(* Logix 5000 project; controller p65 vendor 1 type 14 code 85 rev 20.11; software revision 20.01 *)

TASK ACSTask (continuous, watchdog 500 ms) : Battery, Comm, DCMicroGrid, House01, House02, House03, House04, House05

MODULES
   Local : vendor 1 type 14 code 85 (ICP 4, rev 20.11)
      o : 1756-OB32 (ICP 3, rev 3.1, Output RPI 50 ms)
      i8 : 1756-IF8 (ICP 2, rev 1.1, Input RPI 100 ms)
      i16 : 1756-IF16 (ICP 1, rev 1.1, Input RPI 100 ms)
END_MODULES

VAR_GLOBAL   (* controller tags *)
   BatterybattCurrent : ALIAS FOR REAL00_0;
   BatterybattCurrentHILS : ALIAS FOR plc1_local_3[4];
   Batterybattcurrentoffset : REAL := 2.5261052;
   BatterybattCurrentRaw : ALIAS FOR Local:1:I.Ch4Data;
   BatterybattPower : ALIAS FOR REAL00_1;
   BatterybattVoltage : ALIAS FOR REAL00_2;
   BatterybattVoltageHILS : ALIAS FOR plc1_local_3[5];
   BatterybattVoltageRaw : ALIAS FOR Local:1:I.Ch0Data;
   BatterycanSupplyPower : ALIAS FOR DINT00_22.0;
   Batterycharge : ALIAS FOR REAL00_3;
   BatterychargeCurrent : ALIAS FOR REAL00_4;
   BatterychargeToGo : ALIAS FOR REAL00_5;
   BatterychargingTimer : ALIAS FOR CLTIMER00_0;
   BatterycomputeAddition : ALIAS FOR DINT00_22.7;
   BatterycomputeSubtraction : ALIAS FOR DINT00_22.8;
   BatterydecideToCharge : ALIAS FOR DINT00_22.15;
   BatterydecideToDisconnect : ALIAS FOR DINT00_22.16;
   BatterydeltaCharge : ALIAS FOR REAL00_6;
   BatterydischargeCurrent : ALIAS FOR REAL00_7;
   BatterydischargingTimer : ALIAS FOR CLTIMER00_1;
   BatterydisconnectedTimer : ALIAS FOR CLTIMER00_2;
   Batteryefficiency : ALIAS FOR REAL00_8;
   Batteryfraction : ALIAS FOR REAL00_9;
   BatteryfractionCharged : ALIAS FOR REAL00_10;
   BatteryfractionChargedEstimate : ALIAS FOR REAL00_11;
   BatteryfractionToGo : ALIAS FOR REAL00_12;
   BatteryfullCharge : ALIAS FOR REAL00_13;
   BatteryfullChargeCurrent : ALIAS FOR REAL00_14;
   BatterygeneralTimer : ALIAS FOR CLTIMER00_3;
   BatterygridCurrent : ALIAS FOR REAL00_15;
   BatterygridCurrentabs : REAL := 0.7502556;
   BatterygridCurrentHILS : ALIAS FOR plc1_local_3[2];
   Batterygridcurrentoffset : REAL := 2.529666;
   BatterygridCurrentRaw : ALIAS FOR Local:1:I.Ch5Data;
   BatterygridPower : ALIAS FOR REAL00_16;
   BatterygridVoltage : ALIAS FOR REAL00_17;
   BatterygridVoltageHILS : ALIAS FOR plc1_local_3[3];
   BatterygridVoltageRaw : ALIAS FOR Local:1:I.Ch9Data;
   BatteryintReqCharge : ALIAS FOR DINT00_22.17;
   BatteryintReqDischarge : ALIAS FOR DINT00_22.18;
   BatteryintReqDisconnect : ALIAS FOR DINT00_22.19;
   BatteryisCharging : ALIAS FOR DINT00_22.20;
   BatteryisDischarging : ALIAS FOR DINT00_22.21;
   BatteryisDisconnected : ALIAS FOR DINT00_22.22;
   BatteryisFullyCharged : ALIAS FOR DINT00_22.23;
   BatteryisFunctional : ALIAS FOR DINT00_22.24;
   BatterylastChargingTime : ALIAS FOR DINT00_0;
   BatterylastDischargingTime : ALIAS FOR DINT00_1;
   BatterylastDisconnectedTime : ALIAS FOR DINT00_2;
   BatterylastFractionChargedDelta : ALIAS FOR REAL00_18;
   BatterylastIntReqCharge : ALIAS FOR DINT00_22.25;
   BatterylastIntReqDischarge : ALIAS FOR DINT00_22.26;
   BatterylastIntReqDisconnect : ALIAS FOR DINT00_22.27;
   BatterylowestSOC : ALIAS FOR REAL00_19;
   Batterymultiplier : ALIAS FOR REAL00_20;
   BatterynominalDischargeCurrent : ALIAS FOR REAL00_21;
   BatteryocVoltage : ALIAS FOR REAL00_22;
   BatteryoutOfOperationalRange : ALIAS FOR DINT00_22.28;
   BatterypeukertLessOne : ALIAS FOR REAL00_23;
   Batteryproduct : ALIAS FOR REAL00_24;
   BatteryreqCharge : ALIAS FOR DINT00_22.29;
   BatteryreqDischarge : ALIAS FOR DINT00_22.30;
   BatteryreqDisconnect : ALIAS FOR DINT00_22.31;
   BatteryreqInitialize : ALIAS FOR DINT00_23.0;
   BatterysettlingTimer : ALIAS FOR CLTIMER00_4;
   Batterysoc : ALIAS FOR REAL00_25;
   BatterysocToGo : ALIAS FOR REAL00_26;
   BatterySOCTooLowEventFail : ALIAS FOR DINT00_23.1;
   BatterySOCTooLowEventSuccess : ALIAS FOR DINT00_23.2;
   BatterySOCTooLowFailTimer : ALIAS FOR CLTIMER00_5;
   BatterySOCTooLowInProcess : ALIAS FOR DINT00_23.3;
   BatterySOCTooLowMsg : ALIAS FOR MESSAGE00_0;
   BatterySOCTooLowSuccessTimer : ALIAS FOR CLTIMER00_6;
   BatterytimeSinceLastMeasurement : ALIAS FOR REAL00_27;
   BatterytimeToLowestSOC : ALIAS FOR REAL00_28;
   BatteryunambiguousCommand : ALIAS FOR DINT00_23.4;
   BG_SG_Relay : ALIAS FOR plc1_local_6[1].1;
   CB_SG1_Relay : ALIAS FOR plc1_local_6[1].5;
   CB_SG2_Relay : ALIAS FOR plc1_local_6[1].6;
   CBclose : ALIAS FOR Local:3:O.Data.15;
   CBcloseHILS : ALIAS FOR plc1_local_6[0].14;
   CBcloseProxy : ALIAS FOR DINT00_22.1;
   CBintReqClose : ALIAS FOR DINT00_22.2;
   CBisClosed : ALIAS FOR DINT00_22.3;
   CBisOpen : ALIAS FOR DINT00_22.4;
   CBreqClose : ALIAS FOR DINT00_22.5;
   CBreqOpen : ALIAS FOR DINT00_22.6;
   CF_SG_Relay : ALIAS FOR plc1_local_6[1].7;
   CL1_SG1_Relay : ALIAS FOR plc1_local_6[1].18;
   CL1_SG2_Relay : ALIAS FOR plc1_local_6[1].19;
   CL2_SG1_Relay : ALIAS FOR plc1_local_6[1].20;
   CL2_SG2_Relay : ALIAS FOR plc1_local_6[1].21;
   CL3_SG1_Relay : ALIAS FOR plc1_local_6[1].22;
   CL3_SG2_Relay : ALIAS FOR plc1_local_6[1].23;
   CL4_SG1_Relay : ALIAS FOR plc1_local_6[1].24;
   CL4_SG2_Relay : ALIAS FOR plc1_local_6[1].25;
   CL5_SG1_Relay : ALIAS FOR plc1_local_6[1].26;
   CL5_SG2_Relay : ALIAS FOR plc1_local_6[1].27;
   CLTIMER00_0 : TIMER := (PRE := 1000);
   CLTIMER00_1 : TIMER := (PRE := 1000);
   CLTIMER00_10 : TIMER := (PRE := 3600);
   CLTIMER00_100 : TIMER := (PRE := 1000);
   CLTIMER00_101 : TIMER := (PRE := 5000);
   CLTIMER00_102 : TIMER;
   CLTIMER00_103 : TIMER;
   CLTIMER00_104 : TIMER;
   CLTIMER00_105 : TIMER;
   CLTIMER00_106 : TIMER;
   CLTIMER00_107 : TIMER;
   CLTIMER00_108 : TIMER;
   CLTIMER00_109 : TIMER;
   CLTIMER00_11 : TIMER := (PRE := 3000);
   CLTIMER00_110 : TIMER;
   CLTIMER00_111 : TIMER;
   CLTIMER00_112 : TIMER;
   CLTIMER00_113 : TIMER;
   CLTIMER00_114 : TIMER;
   CLTIMER00_115 : TIMER;
   CLTIMER00_116 : TIMER;
   CLTIMER00_117 : TIMER;
   CLTIMER00_118 : TIMER;
   CLTIMER00_119 : TIMER;
   CLTIMER00_12 : TIMER := (PRE := 10000);
   CLTIMER00_120 : TIMER;
   CLTIMER00_121 : TIMER;
   CLTIMER00_13 : TIMER := (PRE := 5000);
   CLTIMER00_14 : TIMER := (PRE := 10000);
   CLTIMER00_15 : TIMER := (PRE := 500, ACC := 78, EN := 1, TT := 1);
   CLTIMER00_16 : TIMER := (PRE := 5000);
   CLTIMER00_17 : TIMER := (PRE := 3600);
   CLTIMER00_18 : TIMER := (PRE := 3000);
   CLTIMER00_19 : TIMER := (PRE := 10000);
   CLTIMER00_2 : TIMER := (PRE := 1000, ACC := 9, EN := 1, TT := 1);
   CLTIMER00_20 : TIMER := (PRE := 5000);
   CLTIMER00_21 : TIMER := (PRE := 10000);
   CLTIMER00_22 : TIMER := (PRE := 500, ACC := 120, EN := 1, TT := 1);
   CLTIMER00_23 : TIMER := (PRE := 5000);
   CLTIMER00_24 : TIMER := (PRE := 3600);
   CLTIMER00_25 : TIMER := (PRE := 3000);
   CLTIMER00_26 : TIMER := (PRE := 10000);
   CLTIMER00_27 : TIMER := (PRE := 5000);
   CLTIMER00_28 : TIMER := (PRE := 10000);
   CLTIMER00_29 : TIMER := (PRE := 500, ACC := 69, EN := 1, TT := 1);
   CLTIMER00_3 : TIMER := (PRE := 18000, ACC := 9391, EN := 1, TT := 1);
   CLTIMER00_30 : TIMER := (PRE := 5000);
   CLTIMER00_31 : TIMER := (PRE := 3600);
   CLTIMER00_32 : TIMER := (PRE := 3000);
   CLTIMER00_33 : TIMER := (PRE := 10000);
   CLTIMER00_34 : TIMER := (PRE := 5000);
   CLTIMER00_35 : TIMER := (PRE := 10000);
   CLTIMER00_36 : TIMER := (PRE := 500, ACC := 65, EN := 1, TT := 1);
   CLTIMER00_37 : TIMER := (PRE := 5000);
   CLTIMER00_38 : TIMER := (PRE := 3600);
   CLTIMER00_39 : TIMER := (PRE := 3000);
   CLTIMER00_4 : TIMER := (PRE := 300000, ACC := 17125, EN := 1, TT := 1);
   CLTIMER00_40 : TIMER := (PRE := 10000);
   CLTIMER00_41 : TIMER := (PRE := 5000);
   CLTIMER00_42 : TIMER := (PRE := 10000);
   CLTIMER00_43 : TIMER := (PRE := 500, ACC := 121, EN := 1, TT := 1);
   CLTIMER00_44 : TIMER := (PRE := 60000);
   CLTIMER00_45 : TIMER := (PRE := 1000);
   CLTIMER00_46 : TIMER := (PRE := 60000);
   CLTIMER00_47 : TIMER := (PRE := 10000, ACC := 9218, EN := 1, TT := 1);
   CLTIMER00_48 : TIMER := (PRE := 1000000);
   CLTIMER00_49 : TIMER := (PRE := 5000);
   CLTIMER00_5 : TIMER := (PRE := 5000);
   CLTIMER00_50 : TIMER := (PRE := 5000);
   CLTIMER00_51 : TIMER := (PRE := 3600);
   CLTIMER00_52 : TIMER := (PRE := 3000);
   CLTIMER00_53 : TIMER := (PRE := 10000);
   CLTIMER00_54 : TIMER := (PRE := 5000);
   CLTIMER00_55 : TIMER := (PRE := 10000);
   CLTIMER00_56 : TIMER := (PRE := 500, ACC := 26, EN := 1, TT := 1);
   CLTIMER00_57 : TIMER := (PRE := 5000);
   CLTIMER00_58 : TIMER := (PRE := 3600);
   CLTIMER00_59 : TIMER := (PRE := 3000);
   CLTIMER00_6 : TIMER := (PRE := 10000);
   CLTIMER00_60 : TIMER := (PRE := 10000);
   CLTIMER00_61 : TIMER := (PRE := 5000);
   CLTIMER00_62 : TIMER := (PRE := 10000);
   CLTIMER00_63 : TIMER := (PRE := 500, ACC := 62, EN := 1, TT := 1);
   CLTIMER00_64 : TIMER := (PRE := 5000);
   CLTIMER00_65 : TIMER := (PRE := 3600);
   CLTIMER00_66 : TIMER := (PRE := 3000);
   CLTIMER00_67 : TIMER := (PRE := 10000);
   CLTIMER00_68 : TIMER := (PRE := 5000);
   CLTIMER00_69 : TIMER := (PRE := 10000);
   CLTIMER00_7 : TIMER := (PRE := 1000000);
   CLTIMER00_70 : TIMER := (PRE := 500, ACC := 69, EN := 1, TT := 1);
   CLTIMER00_71 : TIMER := (PRE := 5000);
   CLTIMER00_72 : TIMER := (PRE := 3600);
   CLTIMER00_73 : TIMER := (PRE := 3000);
   CLTIMER00_74 : TIMER := (PRE := 10000);
   CLTIMER00_75 : TIMER := (PRE := 5000);
   CLTIMER00_76 : TIMER := (PRE := 10000);
   CLTIMER00_77 : TIMER := (PRE := 500, ACC := 90, EN := 1, TT := 1);
   CLTIMER00_78 : TIMER := (PRE := 5000);
   CLTIMER00_79 : TIMER := (PRE := 3600);
   CLTIMER00_8 : TIMER := (PRE := 5000);
   CLTIMER00_80 : TIMER := (PRE := 3000);
   CLTIMER00_81 : TIMER := (PRE := 10000);
   CLTIMER00_82 : TIMER := (PRE := 5000);
   CLTIMER00_83 : TIMER := (PRE := 10000);
   CLTIMER00_84 : TIMER := (PRE := 500, ACC := 107, EN := 1, TT := 1);
   CLTIMER00_85 : TIMER := (PRE := 60000);
   CLTIMER00_86 : TIMER := (PRE := 1000);
   CLTIMER00_87 : TIMER := (PRE := 60000);
   CLTIMER00_88 : TIMER := (PRE := 10000, ACC := 9235, EN := 1, TT := 1);
   CLTIMER00_89 : TIMER := (PRE := 10000, ACC := 9219, EN := 1, TT := 1);
   CLTIMER00_9 : TIMER := (PRE := 5000);
   CLTIMER00_90 : TIMER := (PRE := 2000);
   CLTIMER00_91 : TIMER := (PRE := 5000);
   CLTIMER00_92 : TIMER := (PRE := 3000);
   CLTIMER00_93 : TIMER := (PRE := 5000);
   CLTIMER00_94 : TIMER := (PRE := 60000);
   CLTIMER00_95 : TIMER := (PRE := 1000);
   CLTIMER00_96 : TIMER := (PRE := 5000);
   CLTIMER00_97 : TIMER := (PRE := 1000);
   CLTIMER00_98 : TIMER := (PRE := 5000);
   CLTIMER00_99 : TIMER := (PRE := 5000);
   Commaccum : ALIAS FOR REAL00_31;
   CommBattempt : ALIAS FOR DINT00_3;
   CommBclose : ALIAS FOR Local:3:O.Data.11;
   CommBcloseHILS : ALIAS FOR plc1_local_6[0].11;
   CommBcloseProxy : ALIAS FOR DINT00_23.12;
   CommBdeadBand : ALIAS FOR REAL00_32;
   CommBfailedToOpen : ALIAS FOR DINT00_23.13;
   CommBintForceOpen : ALIAS FOR DINT00_23.14;
   CommBintReqClose : ALIAS FOR DINT00_23.15;
   CommBisClosed : ALIAS FOR DINT00_23.16;
   CommBisOpen : ALIAS FOR DINT00_23.17;
   CommBmaxAttempts : ALIAS FOR DINT00_4;
   CommBmaxLoadCurrent : ALIAS FOR REAL00_33;
   CommBopenTimer : ALIAS FOR CLTIMER00_7;
   CommBreqClose : ALIAS FOR DINT00_23.18;
   CommBreqOpen : ALIAS FOR DINT00_23.19;
   CommBreqReset : ALIAS FOR DINT00_23.20;
   CommBretriesFailed : ALIAS FOR DINT00_23.21;
   CommBtooMuchCurrent : ALIAS FOR DINT00_23.22;
   CommBunexpectedLowCurrent : ALIAS FOR DINT00_23.23;
   CommcanNotifyUser : ALIAS FOR DINT00_23.24;
   CommcommandChanged : ALIAS FOR DINT00_23.25;
   CommcommandChangedTimer : ALIAS FOR CLTIMER00_8;
   Commcurrent : ALIAS FOR REAL00_34;
   CommcurrentHILS : ALIAS FOR plc1_local_3[8];
   CommcurrentRaw : ALIAS FOR Local:1:I.Ch10Data;
   Commdeadband : ALIAS FOR REAL00_35;
   Commdifference : ALIAS FOR REAL00_36;
   CommfailedToConnect : ALIAS FOR DINT00_23.26;
   CommfailedToDisconnect : ALIAS FOR DINT00_23.27;
   CommintReqConnect : ALIAS FOR DINT00_23.28;
   CommisConnected : ALIAS FOR DINT00_23.29;
   CommisDisconnected : ALIAS FOR DINT00_23.30;
   CommnotificationTimer : ALIAS FOR CLTIMER00_44;
   CommOverCurrentConditionEventFail : ALIAS FOR DINT00_27.13;
   CommOverCurrentConditionEventSuccess : ALIAS FOR DINT00_27.14;
   CommOverCurrentConditionFailTimer : ALIAS FOR CLTIMER00_45;
   CommOverCurrentConditionInProcess : ALIAS FOR DINT00_27.15;
   CommOverCurrentConditionMsg : ALIAS FOR MESSAGE00_11;
   CommOverCurrentConditionSuccessTimer : ALIAS FOR CLTIMER00_46;
   Commpower : ALIAS FOR REAL00_102;
   CommreqConnect : ALIAS FOR DINT00_27.16;
   CommreqDisconnect : ALIAS FOR DINT00_27.17;
   CommsampleNow : ALIAS FOR DINT00_27.18;
   CommsampleTimer : ALIAS FOR CLTIMER00_47;
   Commsuperuser : ALIAS FOR STRING00_5;
   Commtotal : ALIAS FOR REAL00_103;
   CommtotalTooLarge : ALIAS FOR DINT00_27.19;
   CommtotalTooSmall : ALIAS FOR DINT00_27.20;
   CommuserNotified : ALIAS FOR DINT00_27.21;
   Commvoltage : ALIAS FOR REAL00_104;
   CommvoltageHILS : ALIAS FOR plc1_local_3[9];
   CommvoltageRaw : ALIAS FOR Local:2:I.Ch7Data;
   DBclose : ALIAS FOR Local:3:O.Data.14;
   DBcloseHILS : ALIAS FOR plc1_local_6[0].13;
   DBcloseProxy : ALIAS FOR DINT00_22.9;
   DBintReqClose : ALIAS FOR DINT00_22.10;
   DBisClosed : ALIAS FOR DINT00_22.11;
   DBisOpen : ALIAS FOR DINT00_22.12;
   DBreqClose : ALIAS FOR DINT00_22.13;
   DBreqOpen : ALIAS FOR DINT00_22.14;
   DCMicroGridcanNotifyUser : ALIAS FOR DINT00_23.5;
   DCMicroGridfailedToShutdown : ALIAS FOR DINT00_23.6;
   DCMicroGridfailedToStartup : ALIAS FOR DINT00_23.7;
   DCMicroGridinitialPowerRate : ALIAS FOR REAL00_29;
   DCMicroGridisInOperation : ALIAS FOR DINT00_23.8;
   DCMicroGridisShutdown : ALIAS FOR DINT00_23.9;
   DCMicroGridisSimulating : ALIAS FOR DINT00_23.10;
   DCMicroGridisStarted : ALIAS FOR DINT00_23.11;
   DCMicroGridlowestSupportedPriority : ALIAS FOR DINT00_17;
   DCMicroGridmaxPowerRate : ALIAS FOR REAL00_185;
   DCMicroGridmorePowerAvailable : ALIAS FOR DINT00_32.12;
   DCMicroGridnotificationTimer : ALIAS FOR CLTIMER00_94;
   DCMicroGridpowerRate : ALIAS FOR REAL00_186;
   DCMicroGridpowerRateIncrement : REAL := 10.0;
   DCMicroGridrecruitingPhase : ALIAS FOR DINT00_18;
   DCMicroGridreqReset : ALIAS FOR DINT00_32.13;
   DCMicroGridreqShutdown : ALIAS FOR DINT00_32.14;
   DCMicroGridreqStartup : ALIAS FOR DINT00_32.15;
   DCMicroGridResetEventFail : ALIAS FOR DINT00_32.16;
   DCMicroGridResetEventSuccess : ALIAS FOR DINT00_32.17;
   DCMicroGridResetFailTimer : ALIAS FOR CLTIMER00_95;
   DCMicroGridResetInProcess : ALIAS FOR DINT00_32.18;
   DCMicroGridResetMsg : ALIAS FOR MESSAGE00_25;
   DCMicroGridResetSuccessTimer : ALIAS FOR CLTIMER00_96;
   DCMicroGridShutdownEventFail : ALIAS FOR DINT00_32.19;
   DCMicroGridShutdownEventSuccess : ALIAS FOR DINT00_32.20;
   DCMicroGridShutdownFailTimer : ALIAS FOR CLTIMER00_97;
   DCMicroGridShutdownInProcess : ALIAS FOR DINT00_32.21;
   DCMicroGridShutdownMsg : ALIAS FOR MESSAGE00_26;
   DCMicroGridShutdownSuccessTimer : ALIAS FOR CLTIMER00_98;
   DCMicroGridsourcesProvidingExcessPower : ALIAS FOR DINT00_33.7;
   DCMicroGridStartupEventFail : ALIAS FOR DINT00_33.8;
   DCMicroGridStartupEventSuccess : ALIAS FOR DINT00_33.9;
   DCMicroGridStartupFailTimer : ALIAS FOR CLTIMER00_100;
   DCMicroGridStartupInProcess : ALIAS FOR DINT00_33.10;
   DCMicroGridStartupMsg : ALIAS FOR MESSAGE00_27;
   DCMicroGridStartupSuccessTimer : ALIAS FOR CLTIMER00_101;
   DCMicroGridsuperuser : ALIAS FOR STRING00_12;
   DCMicroGridtest : ALIAS FOR REAL00_192;
   DCMicroGridtestout : ALIAS FOR REAL00_193;
   DCMicroGriduserNotified : ALIAS FOR DINT00_33.11;
   DINT00_0 : DINT;
   DINT00_1 : DINT;
   DINT00_10 : DINT;
   DINT00_11 : DINT := 3;
   DINT00_12 : DINT := 10;
   DINT00_13 : DINT := 9;
   DINT00_14 : DINT := 8;
   DINT00_15 : DINT := 7;
   DINT00_16 : DINT := 6;
   DINT00_17 : DINT := 10;
   DINT00_18 : DINT;
   DINT00_19 : DINT;
   DINT00_2 : DINT := 17;
   DINT00_20 : DINT;
   DINT00_21 : DINT;
   DINT00_22 : DINT := -842239919;
   DINT00_23 : DINT := 1225400868;
   DINT00_24 : DINT := 621626516;
   DINT00_25 : DINT := -733396144;
   DINT00_26 : DINT := -1808465328;
   DINT00_27 : DINT := 1086524740;
   DINT00_28 : DINT := 621957153;
   DINT00_29 : DINT := 621363348;
   DINT00_3 : DINT;
   DINT00_30 : DINT := -1811332527;
   DINT00_31 : DINT := 1646596688;
   DINT00_32 : DINT := -1978526464;
   DINT00_33 : DINT := 580;
   DINT00_34 : DINT;
   DINT00_35 : DINT;
   DINT00_4 : DINT := 3;
   DINT00_5 : DINT := 5;
   DINT00_6 : DINT := 4;
   DINT00_7 : DINT := 3;
   DINT00_8 : DINT := 2;
   DINT00_9 : DINT := 1;
   House01accountBalance : ALIAS FOR REAL00_115;
   House01accountDepositRate : ALIAS FOR REAL00_116;
   House01actualGridProvider : ALIAS FOR STRING00_6;
   House01Bclose : ALIAS FOR Local:3:O.Data.0;
   House01BcloseHILS : ALIAS FOR plc1_local_6[0].0;
   House01BcloseProxy : ALIAS FOR DINT00_28.9;
   House01BintReqClose : ALIAS FOR DINT00_28.10;
   House01BisClosed : ALIAS FOR DINT00_28.11;
   House01BisOpen : ALIAS FOR DINT00_28.12;
   House01BreqClose : ALIAS FOR DINT00_28.13;
   House01BreqOpen : ALIAS FOR DINT00_28.14;
   House01commandChanged : ALIAS FOR DINT00_28.15;
   House01commandChangedTimer : ALIAS FOR CLTIMER00_50;
   House01current : ALIAS FOR REAL00_117;
   House01currentHILS : ALIAS FOR plc1_local_2[0];
   House01currentRaw : ALIAS FOR Local:1:I.Ch12Data;
   House01deadband : ALIAS FOR REAL00_118;
   House01depositTimer : ALIAS FOR CLTIMER00_51;
   House01DisconnectPowerEventFail : ALIAS FOR DINT00_28.16;
   House01DisconnectPowerEventSuccess : ALIAS FOR DINT00_28.17;
   House01DisconnectPowerFailTimer : ALIAS FOR CLTIMER00_52;
   House01DisconnectPowerInProcess : ALIAS FOR DINT00_28.18;
   House01DisconnectPowerMsg : ALIAS FOR MESSAGE00_12;
   House01DisconnectPowerSuccessTimer : ALIAS FOR CLTIMER00_53;
   House01failedToConnect : ALIAS FOR DINT00_28.19;
   House01failedToDisconnect : ALIAS FOR DINT00_28.20;
   House01fundsAvailable : ALIAS FOR DINT00_28.21;
   House01incrementToAdd : ALIAS FOR REAL00_119;
   House01incrementToSubtract : ALIAS FOR REAL00_120;
   House01initialAccountBalance : ALIAS FOR REAL00_121;
   House01intReqConnect : ALIAS FOR DINT00_28.22;
   House01isConnected : ALIAS FOR DINT00_28.23;
   House01isDisconnected : ALIAS FOR DINT00_28.24;
   House01minBalance : ALIAS FOR REAL00_122;
   House01minBalanceToReconnect : ALIAS FOR REAL00_123;
   House01minTime : ALIAS FOR REAL00_124;
   House01powerRate : ALIAS FOR REAL00_125;
   House01powerRateMax : REAL := 40.0;
   House01priority : ALIAS FOR DINT00_12;
   House01PurchasePowerEventFail : ALIAS FOR DINT00_28.25;
   House01PurchasePowerEventSuccess : ALIAS FOR DINT00_28.26;
   House01PurchasePowerFailTimer : ALIAS FOR CLTIMER00_54;
   House01PurchasePowerInProcess : ALIAS FOR DINT00_28.27;
   House01PurchasePowerMsg : ALIAS FOR MESSAGE00_13;
   House01PurchasePowerSuccessTimer : ALIAS FOR CLTIMER00_55;
   House01reqConnect : ALIAS FOR DINT00_28.28;
   House01reqDisconnect : ALIAS FOR DINT00_28.29;
   House01runningOut : ALIAS FOR DINT00_28.30;
   House01spendingRate : ALIAS FOR REAL00_126;
   House01timeRemaining : ALIAS FOR REAL00_127;
   House01usageTimer : ALIAS FOR CLTIMER00_56;
   House02accountBalance : ALIAS FOR REAL00_128;
   House02accountDepositRate : ALIAS FOR REAL00_129;
   House02actualGridProvider : ALIAS FOR STRING00_7;
   House02Bclose : ALIAS FOR Local:3:O.Data.1;
   House02BcloseHILS : ALIAS FOR plc1_local_6[0].1;
   House02BcloseProxy : ALIAS FOR DINT00_28.31;
   House02BintReqClose : ALIAS FOR DINT00_29.0;
   House02BisClosed : ALIAS FOR DINT00_29.1;
   House02BisOpen : ALIAS FOR DINT00_29.2;
   House02BreqClose : ALIAS FOR DINT00_29.3;
   House02BreqOpen : ALIAS FOR DINT00_29.4;
   House02commandChanged : ALIAS FOR DINT00_29.5;
   House02commandChangedTimer : ALIAS FOR CLTIMER00_57;
   House02current : ALIAS FOR REAL00_130;
   House02currentHILS : ALIAS FOR plc1_local_2[1];
   House02currentRaw : ALIAS FOR Local:1:I.Ch13Data;
   House02deadband : ALIAS FOR REAL00_131;
   House02depositTimer : ALIAS FOR CLTIMER00_58;
   House02DisconnectPowerEventFail : ALIAS FOR DINT00_29.6;
   House02DisconnectPowerEventSuccess : ALIAS FOR DINT00_29.7;
   House02DisconnectPowerFailTimer : ALIAS FOR CLTIMER00_59;
   House02DisconnectPowerInProcess : ALIAS FOR DINT00_29.8;
   House02DisconnectPowerMsg : ALIAS FOR MESSAGE00_14;
   House02DisconnectPowerSuccessTimer : ALIAS FOR CLTIMER00_60;
   House02failedToConnect : ALIAS FOR DINT00_29.9;
   House02failedToDisconnect : ALIAS FOR DINT00_29.10;
   House02fundsAvailable : ALIAS FOR DINT00_29.11;
   House02incrementToAdd : ALIAS FOR REAL00_132;
   House02incrementToSubtract : ALIAS FOR REAL00_133;
   House02initialAccountBalance : ALIAS FOR REAL00_134;
   House02intReqConnect : ALIAS FOR DINT00_29.12;
   House02isConnected : ALIAS FOR DINT00_29.13;
   House02isDisconnected : ALIAS FOR DINT00_29.14;
   House02minBalance : ALIAS FOR REAL00_135;
   House02minBalanceToReconnect : ALIAS FOR REAL00_136;
   House02minTime : ALIAS FOR REAL00_137;
   House02powerRate : ALIAS FOR REAL00_138;
   House02powerRateMax : REAL := 40.0;
   House02priority : ALIAS FOR DINT00_13;
   House02PurchasePowerEventFail : ALIAS FOR DINT00_29.15;
   House02PurchasePowerEventSuccess : ALIAS FOR DINT00_29.16;
   House02PurchasePowerFailTimer : ALIAS FOR CLTIMER00_61;
   House02PurchasePowerInProcess : ALIAS FOR DINT00_29.17;
   House02PurchasePowerMsg : ALIAS FOR MESSAGE00_15;
   House02PurchasePowerSuccessTimer : ALIAS FOR CLTIMER00_62;
   House02reqConnect : ALIAS FOR DINT00_29.18;
   House02reqDisconnect : ALIAS FOR DINT00_29.19;
   House02runningOut : ALIAS FOR DINT00_29.20;
   House02spendingRate : ALIAS FOR REAL00_139;
   House02timeRemaining : ALIAS FOR REAL00_140;
   House02usageTimer : ALIAS FOR CLTIMER00_63;
   House03accountBalance : ALIAS FOR REAL00_141;
   House03accountDepositRate : ALIAS FOR REAL00_142;
   House03actualGridProvider : ALIAS FOR STRING00_8;
   House03Bclose : ALIAS FOR Local:3:O.Data.2;
   House03BcloseHILS : ALIAS FOR plc1_local_6[0].2;
   House03BcloseProxy : ALIAS FOR DINT00_29.21;
   House03BintReqClose : ALIAS FOR DINT00_29.22;
   House03BisClosed : ALIAS FOR DINT00_29.23;
   House03BisOpen : ALIAS FOR DINT00_29.24;
   House03BreqClose : ALIAS FOR DINT00_29.25;
   House03BreqOpen : ALIAS FOR DINT00_29.26;
   House03commandChanged : ALIAS FOR DINT00_29.27;
   House03commandChangedTimer : ALIAS FOR CLTIMER00_64;
   House03current : ALIAS FOR REAL00_143;
   House03currentHILS : ALIAS FOR plc1_local_2[2];
   House03currentRaw : ALIAS FOR Local:1:I.Ch14Data;
   House03deadband : ALIAS FOR REAL00_144;
   House03depositTimer : ALIAS FOR CLTIMER00_65;
   House03DisconnectPowerEventFail : ALIAS FOR DINT00_29.28;
   House03DisconnectPowerEventSuccess : ALIAS FOR DINT00_29.29;
   House03DisconnectPowerFailTimer : ALIAS FOR CLTIMER00_66;
   House03DisconnectPowerInProcess : ALIAS FOR DINT00_29.30;
   House03DisconnectPowerMsg : ALIAS FOR MESSAGE00_16;
   House03DisconnectPowerSuccessTimer : ALIAS FOR CLTIMER00_67;
   House03failedToConnect : ALIAS FOR DINT00_29.31;
   House03failedToDisconnect : ALIAS FOR DINT00_30.0;
   House03fundsAvailable : ALIAS FOR DINT00_30.1;
   House03incrementToAdd : ALIAS FOR REAL00_145;
   House03incrementToSubtract : ALIAS FOR REAL00_146;
   House03initialAccountBalance : ALIAS FOR REAL00_147;
   House03intReqConnect : ALIAS FOR DINT00_30.2;
   House03isConnected : ALIAS FOR DINT00_30.3;
   House03isDisconnected : ALIAS FOR DINT00_30.4;
   House03minBalance : ALIAS FOR REAL00_148;
   House03minBalanceToReconnect : ALIAS FOR REAL00_149;
   House03minTime : ALIAS FOR REAL00_150;
   House03powerRate : ALIAS FOR REAL00_151;
   House03powerRateMax : REAL := 30.0;
   House03priority : ALIAS FOR DINT00_14;
   House03PurchasePowerEventFail : ALIAS FOR DINT00_30.5;
   House03PurchasePowerEventSuccess : ALIAS FOR DINT00_30.6;
   House03PurchasePowerFailTimer : ALIAS FOR CLTIMER00_68;
   House03PurchasePowerInProcess : ALIAS FOR DINT00_30.7;
   House03PurchasePowerMsg : ALIAS FOR MESSAGE00_17;
   House03PurchasePowerSuccessTimer : ALIAS FOR CLTIMER00_69;
   House03reqConnect : ALIAS FOR DINT00_30.8;
   House03reqDisconnect : ALIAS FOR DINT00_30.9;
   House03runningOut : ALIAS FOR DINT00_30.10;
   House03spendingRate : ALIAS FOR REAL00_152;
   House03timeRemaining : ALIAS FOR REAL00_153;
   House03usageTimer : ALIAS FOR CLTIMER00_70;
   House04accountBalance : ALIAS FOR REAL00_154;
   House04accountDepositRate : ALIAS FOR REAL00_155;
   House04actualGridProvider : ALIAS FOR STRING00_9;
   House04Bclose : ALIAS FOR Local:3:O.Data.3;
   House04BcloseHILS : ALIAS FOR plc1_local_6[0].3;
   House04BcloseProxy : ALIAS FOR DINT00_30.11;
   House04BintReqClose : ALIAS FOR DINT00_30.12;
   House04BisClosed : ALIAS FOR DINT00_30.13;
   House04BisOpen : ALIAS FOR DINT00_30.14;
   House04BreqClose : ALIAS FOR DINT00_30.15;
   House04BreqOpen : ALIAS FOR DINT00_30.16;
   House04commandChanged : ALIAS FOR DINT00_30.17;
   House04commandChangedTimer : ALIAS FOR CLTIMER00_71;
   House04current : ALIAS FOR REAL00_156;
   House04currentHILS : ALIAS FOR plc1_local_2[3];
   House04currentRaw : ALIAS FOR Local:1:I.Ch15Data;
   House04deadband : ALIAS FOR REAL00_157;
   House04depositTimer : ALIAS FOR CLTIMER00_72;
   House04DisconnectPowerEventFail : ALIAS FOR DINT00_30.18;
   House04DisconnectPowerEventSuccess : ALIAS FOR DINT00_30.19;
   House04DisconnectPowerFailTimer : ALIAS FOR CLTIMER00_73;
   House04DisconnectPowerInProcess : ALIAS FOR DINT00_30.20;
   House04DisconnectPowerMsg : ALIAS FOR MESSAGE00_18;
   House04DisconnectPowerSuccessTimer : ALIAS FOR CLTIMER00_74;
   House04failedToConnect : ALIAS FOR DINT00_30.21;
   House04failedToDisconnect : ALIAS FOR DINT00_30.22;
   House04fundsAvailable : ALIAS FOR DINT00_30.23;
   House04incrementToAdd : ALIAS FOR REAL00_158;
   House04incrementToSubtract : ALIAS FOR REAL00_159;
   House04initialAccountBalance : ALIAS FOR REAL00_160;
   House04intReqConnect : ALIAS FOR DINT00_30.24;
   House04isConnected : ALIAS FOR DINT00_30.25;
   House04isDisconnected : ALIAS FOR DINT00_30.26;
   House04minBalance : ALIAS FOR REAL00_161;
   House04minBalanceToReconnect : ALIAS FOR REAL00_162;
   House04minTime : ALIAS FOR REAL00_163;
   House04poweRateMax : REAL;
   House04powerRate : ALIAS FOR REAL00_164;
   House04powerRateMax : REAL := 30.0;
   House04priority : ALIAS FOR DINT00_15;
   House04PurchasePowerEventFail : ALIAS FOR DINT00_30.27;
   House04PurchasePowerEventSuccess : ALIAS FOR DINT00_30.28;
   House04PurchasePowerFailTimer : ALIAS FOR CLTIMER00_75;
   House04PurchasePowerInProcess : ALIAS FOR DINT00_30.29;
   House04PurchasePowerMsg : ALIAS FOR MESSAGE00_19;
   House04PurchasePowerSuccessTimer : ALIAS FOR CLTIMER00_76;
   House04reqConnect : ALIAS FOR DINT00_30.30;
   House04reqDisconnect : ALIAS FOR DINT00_30.31;
   House04runningOut : ALIAS FOR DINT00_31.0;
   House04spendingRate : ALIAS FOR REAL00_165;
   House04timeRemaining : ALIAS FOR REAL00_166;
   House04usageTimer : ALIAS FOR CLTIMER00_77;
   House05accountBalance : ALIAS FOR REAL00_167;
   House05accountDepositRate : ALIAS FOR REAL00_168;
   House05actualGridProvider : ALIAS FOR STRING00_10;
   House05Bclose : ALIAS FOR Local:3:O.Data.4;
   House05BcloseHILS : ALIAS FOR plc1_local_6[0].4;
   House05BcloseProxy : ALIAS FOR DINT00_31.1;
   House05BintReqClose : ALIAS FOR DINT00_31.2;
   House05BisClosed : ALIAS FOR DINT00_31.3;
   House05BisOpen : ALIAS FOR DINT00_31.4;
   House05BreqClose : ALIAS FOR DINT00_31.5;
   House05BreqOpen : ALIAS FOR DINT00_31.6;
   House05commandChanged : ALIAS FOR DINT00_31.7;
   House05commandChangedTimer : ALIAS FOR CLTIMER00_78;
   House05current : ALIAS FOR REAL00_169;
   House05currentHILS : ALIAS FOR plc1_local_2[4];
   House05currentRaw : ALIAS FOR Local:2:I.Ch0Data;
   House05deadband : ALIAS FOR REAL00_170;
   House05depositTimer : ALIAS FOR CLTIMER00_79;
   House05DisconnectPowerEventFail : ALIAS FOR DINT00_31.8;
   House05DisconnectPowerEventSuccess : ALIAS FOR DINT00_31.9;
   House05DisconnectPowerFailTimer : ALIAS FOR CLTIMER00_80;
   House05DisconnectPowerInProcess : ALIAS FOR DINT00_31.10;
   House05DisconnectPowerMsg : ALIAS FOR MESSAGE00_20;
   House05DisconnectPowerSuccessTimer : ALIAS FOR CLTIMER00_81;
   House05failedToConnect : ALIAS FOR DINT00_31.11;
   House05failedToDisconnect : ALIAS FOR DINT00_31.12;
   House05fundsAvailable : ALIAS FOR DINT00_31.13;
   House05incrementToAdd : ALIAS FOR REAL00_171;
   House05incrementToSubtract : ALIAS FOR REAL00_172;
   House05initialAccountBalance : ALIAS FOR REAL00_173;
   House05intReqConnect : ALIAS FOR DINT00_31.14;
   House05isConnected : ALIAS FOR DINT00_31.15;
   House05isDisconnected : ALIAS FOR DINT00_31.16;
   House05minBalance : ALIAS FOR REAL00_174;
   House05minBalanceToReconnect : ALIAS FOR REAL00_175;
   House05minTime : ALIAS FOR REAL00_176;
   House05powerRate : ALIAS FOR REAL00_177;
   House05powerRateMax : REAL := 60.0;
   House05priority : ALIAS FOR DINT00_16;
   House05PurchasePowerEventFail : ALIAS FOR DINT00_31.17;
   House05PurchasePowerEventSuccess : ALIAS FOR DINT00_31.18;
   House05PurchasePowerFailTimer : ALIAS FOR CLTIMER00_82;
   House05PurchasePowerInProcess : ALIAS FOR DINT00_31.19;
   House05PurchasePowerMsg : ALIAS FOR MESSAGE00_21;
   House05PurchasePowerSuccessTimer : ALIAS FOR CLTIMER00_83;
   House05reqConnect : ALIAS FOR DINT00_31.20;
   House05reqDisconnect : ALIAS FOR DINT00_31.21;
   House05runningOut : ALIAS FOR DINT00_31.22;
   House05spendingRate : ALIAS FOR REAL00_178;
   House05timeRemaining : ALIAS FOR REAL00_179;
   House05usageTimer : ALIAS FOR CLTIMER00_84;
   LastSolar_Power : REAL;
   Load01accountBalance : ALIAS FOR REAL00_37;
   Load01accountDepositRate : ALIAS FOR REAL00_38;
   Load01actualGridProvider : ALIAS FOR STRING00_0;
   Load01Bclose : ALIAS FOR Local:3:O.Data.5;
   Load01BcloseHILS : ALIAS FOR plc1_local_6[0].5;
   Load01BcloseProxy : ALIAS FOR DINT00_23.31;
   Load01BintReqClose : ALIAS FOR DINT00_24.0;
   Load01BisClosed : ALIAS FOR DINT00_24.1;
   Load01BisOpen : ALIAS FOR DINT00_24.2;
   Load01BreqClose : ALIAS FOR DINT00_24.3;
   Load01BreqOpen : ALIAS FOR DINT00_24.4;
   Load01commandChanged : ALIAS FOR DINT00_24.5;
   Load01commandChangedTimer : ALIAS FOR CLTIMER00_9;
   Load01current : ALIAS FOR REAL00_39;
   Load01currentHILS : ALIAS FOR plc1_local_2[5];
   Load01currentRaw : ALIAS FOR Local:2:I.Ch2Data;
   Load01deadband : ALIAS FOR REAL00_40;
   Load01depositTimer : ALIAS FOR CLTIMER00_10;
   Load01DisconnectPowerEventFail : ALIAS FOR DINT00_24.6;
   Load01DisconnectPowerEventSuccess : ALIAS FOR DINT00_24.7;
   Load01DisconnectPowerFailTimer : ALIAS FOR CLTIMER00_11;
   Load01DisconnectPowerInProcess : ALIAS FOR DINT00_24.8;
   Load01DisconnectPowerMsg : ALIAS FOR MESSAGE00_1;
   Load01DisconnectPowerSuccessTimer : ALIAS FOR CLTIMER00_12;
   Load01failedToConnect : ALIAS FOR DINT00_24.9;
   Load01failedToDisconnect : ALIAS FOR DINT00_24.10;
   Load01fundsAvailable : ALIAS FOR DINT00_24.11;
   Load01incrementToAdd : ALIAS FOR REAL00_41;
   Load01incrementToSubtract : ALIAS FOR REAL00_42;
   Load01initialAccountBalance : ALIAS FOR REAL00_43;
   Load01intReqConnect : ALIAS FOR DINT00_24.12;
   Load01isConnected : ALIAS FOR DINT00_24.13;
   Load01isDisconnected : ALIAS FOR DINT00_24.14;
   Load01minBalance : ALIAS FOR REAL00_44;
   Load01minBalanceToReconnect : ALIAS FOR REAL00_45;
   Load01minTime : ALIAS FOR REAL00_46;
   Load01powerRate : ALIAS FOR REAL00_47;
   Load01powerRateMax : REAL := 80.0;
   Load01priority : ALIAS FOR DINT00_5;
   Load01PurchasePowerEventFail : ALIAS FOR DINT00_24.15;
   Load01PurchasePowerEventSuccess : ALIAS FOR DINT00_24.16;
   Load01PurchasePowerFailTimer : ALIAS FOR CLTIMER00_13;
   Load01PurchasePowerInProcess : ALIAS FOR DINT00_24.17;
   Load01PurchasePowerMsg : ALIAS FOR MESSAGE00_2;
   Load01PurchasePowerSuccessTimer : ALIAS FOR CLTIMER00_14;
   Load01reqConnect : ALIAS FOR DINT00_24.18;
   Load01reqDisconnect : ALIAS FOR DINT00_24.19;
   Load01runningOut : ALIAS FOR DINT00_24.20;
   Load01spendingRate : ALIAS FOR REAL00_48;
   Load01timeRemaining : ALIAS FOR REAL00_49;
   Load01usageTimer : ALIAS FOR CLTIMER00_15;
   Load02accountBalance : ALIAS FOR REAL00_50;
   Load02accountDepositRate : ALIAS FOR REAL00_51;
   Load02actualGridProvider : ALIAS FOR STRING00_1;
   Load02Bclose : ALIAS FOR Local:3:O.Data.6;
   Load02BcloseHILS : ALIAS FOR plc1_local_6[0].6;
   Load02BcloseProxy : ALIAS FOR DINT00_24.21;
   Load02BintReqClose : ALIAS FOR DINT00_24.22;
   Load02BisClosed : ALIAS FOR DINT00_24.23;
   Load02BisOpen : ALIAS FOR DINT00_24.24;
   Load02BreqClose : ALIAS FOR DINT00_24.25;
   Load02BreqOpen : ALIAS FOR DINT00_24.26;
   Load02commandChanged : ALIAS FOR DINT00_24.27;
   Load02commandChangedTimer : ALIAS FOR CLTIMER00_16;
   Load02current : ALIAS FOR REAL00_52;
   Load02currentHILS : ALIAS FOR plc1_local_2[6];
   Load02currentRaw : ALIAS FOR Local:2:I.Ch3Data;
   Load02deadband : ALIAS FOR REAL00_53;
   Load02depositTimer : ALIAS FOR CLTIMER00_17;
   Load02DisconnectPowerEventFail : ALIAS FOR DINT00_24.28;
   Load02DisconnectPowerEventSuccess : ALIAS FOR DINT00_24.29;
   Load02DisconnectPowerFailTimer : ALIAS FOR CLTIMER00_18;
   Load02DisconnectPowerInProcess : ALIAS FOR DINT00_24.30;
   Load02DisconnectPowerMsg : ALIAS FOR MESSAGE00_3;
   Load02DisconnectPowerSuccessTimer : ALIAS FOR CLTIMER00_19;
   Load02failedToConnect : ALIAS FOR DINT00_24.31;
   Load02failedToDisconnect : ALIAS FOR DINT00_25.0;
   Load02fundsAvailable : ALIAS FOR DINT00_25.1;
   Load02incrementToAdd : ALIAS FOR REAL00_54;
   Load02incrementToSubtract : ALIAS FOR REAL00_55;
   Load02initialAccountBalance : ALIAS FOR REAL00_56;
   Load02intReqConnect : ALIAS FOR DINT00_25.2;
   Load02isConnected : ALIAS FOR DINT00_25.3;
   Load02isDisconnected : ALIAS FOR DINT00_25.4;
   Load02minBalance : ALIAS FOR REAL00_57;
   Load02minBalanceToReconnect : ALIAS FOR REAL00_58;
   Load02minTime : ALIAS FOR REAL00_59;
   Load02powerRate : ALIAS FOR REAL00_60;
   Load02powerRateMax : REAL := 110.0;
   Load02priority : ALIAS FOR DINT00_6;
   Load02PurchasePowerEventFail : ALIAS FOR DINT00_25.5;
   Load02PurchasePowerEventSuccess : ALIAS FOR DINT00_25.6;
   Load02PurchasePowerFailTimer : ALIAS FOR CLTIMER00_20;
   Load02PurchasePowerInProcess : ALIAS FOR DINT00_25.7;
   Load02PurchasePowerMsg : ALIAS FOR MESSAGE00_4;
   Load02PurchasePowerSuccessTimer : ALIAS FOR CLTIMER00_21;
   Load02reqConnect : ALIAS FOR DINT00_25.8;
   Load02reqDisconnect : ALIAS FOR DINT00_25.9;
   Load02runningOut : ALIAS FOR DINT00_25.10;
   Load02spendingRate : ALIAS FOR REAL00_61;
   Load02timeRemaining : ALIAS FOR REAL00_62;
   Load02usageTimer : ALIAS FOR CLTIMER00_22;
   Load03accountBalance : ALIAS FOR REAL00_63;
   Load03accountDepositRate : ALIAS FOR REAL00_64;
   Load03actualGridProvider : ALIAS FOR STRING00_2;
   Load03Bclose : ALIAS FOR Local:3:O.Data.7;
   Load03BcloseHILS : ALIAS FOR plc1_local_6[0].7;
   Load03BcloseProxy : ALIAS FOR DINT00_25.11;
   Load03BintReqClose : ALIAS FOR DINT00_25.12;
   Load03BisClosed : ALIAS FOR DINT00_25.13;
   Load03BisOpen : ALIAS FOR DINT00_25.14;
   Load03BreqClose : ALIAS FOR DINT00_25.15;
   Load03BreqOpen : ALIAS FOR DINT00_25.16;
   Load03commandChanged : ALIAS FOR DINT00_25.17;
   Load03commandChangedTimer : ALIAS FOR CLTIMER00_23;
   Load03current : ALIAS FOR REAL00_65;
   Load03currentHILS : ALIAS FOR plc1_local_2[7];
   Load03currentRaw : ALIAS FOR Local:2:I.Ch4Data;
   Load03deadband : ALIAS FOR REAL00_66;
   Load03depositTimer : ALIAS FOR CLTIMER00_24;
   Load03DisconnectPowerEventFail : ALIAS FOR DINT00_25.18;
   Load03DisconnectPowerEventSuccess : ALIAS FOR DINT00_25.19;
   Load03DisconnectPowerFailTimer : ALIAS FOR CLTIMER00_25;
   Load03DisconnectPowerInProcess : ALIAS FOR DINT00_25.20;
   Load03DisconnectPowerMsg : ALIAS FOR MESSAGE00_5;
   Load03DisconnectPowerSuccessTimer : ALIAS FOR CLTIMER00_26;
   Load03failedToConnect : ALIAS FOR DINT00_25.21;
   Load03failedToDisconnect : ALIAS FOR DINT00_25.22;
   Load03fundsAvailable : ALIAS FOR DINT00_25.23;
   Load03incrementToAdd : ALIAS FOR REAL00_67;
   Load03incrementToSubtract : ALIAS FOR REAL00_68;
   Load03initialAccountBalance : ALIAS FOR REAL00_69;
   Load03intReqConnect : ALIAS FOR DINT00_25.24;
   Load03isConnected : ALIAS FOR DINT00_25.25;
   Load03isDisconnected : ALIAS FOR DINT00_25.26;
   Load03minBalance : ALIAS FOR REAL00_70;
   Load03minBalanceToReconnect : ALIAS FOR REAL00_71;
   Load03minTime : ALIAS FOR REAL00_72;
   Load03powerRate : ALIAS FOR REAL00_73;
   Load03powerRateMax : REAL := 110.0;
   Load03priority : ALIAS FOR DINT00_7;
   Load03PurchasePowerEventFail : ALIAS FOR DINT00_25.27;
   Load03PurchasePowerEventSuccess : ALIAS FOR DINT00_25.28;
   Load03PurchasePowerFailTimer : ALIAS FOR CLTIMER00_27;
   Load03PurchasePowerInProcess : ALIAS FOR DINT00_25.29;
   Load03PurchasePowerMsg : ALIAS FOR MESSAGE00_6;
   Load03PurchasePowerSuccessTimer : ALIAS FOR CLTIMER00_28;
   Load03reqConnect : ALIAS FOR DINT00_25.30;
   Load03reqDisconnect : ALIAS FOR DINT00_25.31;
   Load03runningOut : ALIAS FOR DINT00_26.0;
   Load03spendingRate : ALIAS FOR REAL00_74;
   Load03timeRemaining : ALIAS FOR REAL00_75;
   Load03usageTimer : ALIAS FOR CLTIMER00_29;
   Load04accountBalance : ALIAS FOR REAL00_76;
   Load04accountDepositRate : ALIAS FOR REAL00_77;
   Load04actualGridProvider : ALIAS FOR STRING00_3;
   Load04Bclose : ALIAS FOR Local:3:O.Data.8;
   Load04BcloseHILS : ALIAS FOR plc1_local_6[0].8;
   Load04BcloseProxy : ALIAS FOR DINT00_26.1;
   Load04BintReqClose : ALIAS FOR DINT00_26.2;
   Load04BisClosed : ALIAS FOR DINT00_26.3;
   Load04BisOpen : ALIAS FOR DINT00_26.4;
   Load04BreqClose : ALIAS FOR DINT00_26.5;
   Load04BreqOpen : ALIAS FOR DINT00_26.6;
   Load04commandChanged : ALIAS FOR DINT00_26.7;
   Load04commandChangedTimer : ALIAS FOR CLTIMER00_30;
   Load04current : ALIAS FOR REAL00_78;
   Load04currentHILS : ALIAS FOR plc1_local_2[8];
   Load04currentRaw : ALIAS FOR Local:2:I.Ch5Data;
   Load04deadband : ALIAS FOR REAL00_79;
   Load04depositTimer : ALIAS FOR CLTIMER00_31;
   Load04DisconnectPowerEventFail : ALIAS FOR DINT00_26.8;
   Load04DisconnectPowerEventSuccess : ALIAS FOR DINT00_26.9;
   Load04DisconnectPowerFailTimer : ALIAS FOR CLTIMER00_32;
   Load04DisconnectPowerInProcess : ALIAS FOR DINT00_26.10;
   Load04DisconnectPowerMsg : ALIAS FOR MESSAGE00_7;
   Load04DisconnectPowerSuccessTimer : ALIAS FOR CLTIMER00_33;
   Load04failedToConnect : ALIAS FOR DINT00_26.11;
   Load04failedToDisconnect : ALIAS FOR DINT00_26.12;
   Load04fundsAvailable : ALIAS FOR DINT00_26.13;
   Load04incrementToAdd : ALIAS FOR REAL00_80;
   Load04incrementToSubtract : ALIAS FOR REAL00_81;
   Load04initialAccountBalance : ALIAS FOR REAL00_82;
   Load04intReqConnect : ALIAS FOR DINT00_26.14;
   Load04isConnected : ALIAS FOR DINT00_26.15;
   Load04isDisconnected : ALIAS FOR DINT00_26.16;
   Load04minBalance : ALIAS FOR REAL00_83;
   Load04minBalanceToReconnect : ALIAS FOR REAL00_84;
   Load04minTime : ALIAS FOR REAL00_85;
   Load04powerRate : ALIAS FOR REAL00_86;
   Load04powerRateMax : REAL := 110.0;
   Load04priority : ALIAS FOR DINT00_8;
   Load04PurchasePowerEventFail : ALIAS FOR DINT00_26.17;
   Load04PurchasePowerEventSuccess : ALIAS FOR DINT00_26.18;
   Load04PurchasePowerFailTimer : ALIAS FOR CLTIMER00_34;
   Load04PurchasePowerInProcess : ALIAS FOR DINT00_26.19;
   Load04PurchasePowerMsg : ALIAS FOR MESSAGE00_8;
   Load04PurchasePowerSuccessTimer : ALIAS FOR CLTIMER00_35;
   Load04reqConnect : ALIAS FOR DINT00_26.20;
   Load04reqDisconnect : ALIAS FOR DINT00_26.21;
   Load04runningOut : ALIAS FOR DINT00_26.22;
   Load04spendingRate : ALIAS FOR REAL00_87;
   Load04timeRemaining : ALIAS FOR REAL00_88;
   Load04usageTimer : ALIAS FOR CLTIMER00_36;
   Load05accountBalance : ALIAS FOR REAL00_89;
   Load05accountDepositRate : ALIAS FOR REAL00_90;
   Load05actualGridProvider : ALIAS FOR STRING00_4;
   Load05Bclose : ALIAS FOR Local:3:O.Data.9;
   Load05BcloseHILS : ALIAS FOR plc1_local_6[0].9;
   Load05BcloseProxy : ALIAS FOR DINT00_26.23;
   Load05BintReqClose : ALIAS FOR DINT00_26.24;
   Load05BisClosed : ALIAS FOR DINT00_26.25;
   Load05BisOpen : ALIAS FOR DINT00_26.26;
   Load05BreqClose : ALIAS FOR DINT00_26.27;
   Load05BreqOpen : ALIAS FOR DINT00_26.28;
   Load05commandChanged : ALIAS FOR DINT00_26.29;
   Load05commandChangedTimer : ALIAS FOR CLTIMER00_37;
   Load05current : ALIAS FOR REAL00_91;
   Load05currentHILS : ALIAS FOR plc1_local_2[9];
   Load05currentRaw : ALIAS FOR Local:2:I.Ch6Data;
   Load05deadband : ALIAS FOR REAL00_92;
   Load05depositTimer : ALIAS FOR CLTIMER00_38;
   Load05DisconnectPowerEventFail : ALIAS FOR DINT00_26.30;
   Load05DisconnectPowerEventSuccess : ALIAS FOR DINT00_26.31;
   Load05DisconnectPowerFailTimer : ALIAS FOR CLTIMER00_39;
   Load05DisconnectPowerInProcess : ALIAS FOR DINT00_27.0;
   Load05DisconnectPowerMsg : ALIAS FOR MESSAGE00_9;
   Load05DisconnectPowerSuccessTimer : ALIAS FOR CLTIMER00_40;
   Load05failedToConnect : ALIAS FOR DINT00_27.1;
   Load05failedToDisconnect : ALIAS FOR DINT00_27.2;
   Load05fundsAvailable : ALIAS FOR DINT00_27.3;
   Load05incrementToAdd : ALIAS FOR REAL00_93;
   Load05incrementToSubtract : ALIAS FOR REAL00_94;
   Load05initialAccountBalance : ALIAS FOR REAL00_95;
   Load05intReqConnect : ALIAS FOR DINT00_27.4;
   Load05isConnected : ALIAS FOR DINT00_27.5;
   Load05isDisconnected : ALIAS FOR DINT00_27.6;
   Load05minBalance : ALIAS FOR REAL00_96;
   Load05minBalanceToReconnect : ALIAS FOR REAL00_97;
   Load05minTime : ALIAS FOR REAL00_98;
   Load05powerRate : ALIAS FOR REAL00_99;
   Load05powerRateMax : REAL := 110.0;
   Load05priority : ALIAS FOR DINT00_9;
   Load05PurchasePowerEventFail : ALIAS FOR DINT00_27.7;
   Load05PurchasePowerEventSuccess : ALIAS FOR DINT00_27.8;
   Load05PurchasePowerFailTimer : ALIAS FOR CLTIMER00_41;
   Load05PurchasePowerInProcess : ALIAS FOR DINT00_27.9;
   Load05PurchasePowerMsg : ALIAS FOR MESSAGE00_10;
   Load05PurchasePowerSuccessTimer : ALIAS FOR CLTIMER00_42;
   Load05reqConnect : ALIAS FOR DINT00_27.10;
   Load05reqDisconnect : ALIAS FOR DINT00_27.11;
   Load05runningOut : ALIAS FOR DINT00_27.12;
   Load05spendingRate : ALIAS FOR REAL00_100;
   Load05timeRemaining : ALIAS FOR REAL00_101;
   Load05usageTimer : ALIAS FOR CLTIMER00_43;
   Loadsaccum : ALIAS FOR REAL00_30;
   Loadscurrent : ALIAS FOR REAL00_105;
   LoadscurrentHILS : ALIAS FOR plc1_local_5[0];
   LoadscurrentRaw : ALIAS FOR Local:1:I.Ch6Data;
   Loadsdifference : ALIAS FOR REAL00_106;
   LoadslastLowVoltage : ALIAS FOR DINT00_27.22;
   LoadslowVoltage : ALIAS FOR DINT00_27.23;
   LoadslowVoltageBound : ALIAS FOR REAL00_107;
   Loadspower : ALIAS FOR REAL00_108;
   Loadsrecovered : ALIAS FOR DINT00_27.24;
   LoadssampleNow : ALIAS FOR DINT00_32.3;
   LoadssampleTimer : ALIAS FOR CLTIMER00_89;
   Loadstotal : ALIAS FOR REAL00_183;
   LoadstotalTooLarge : ALIAS FOR DINT00_32.4;
   LoadstotalTooSmall : ALIAS FOR DINT00_32.5;
   Loadsvoltage : ALIAS FOR REAL00_184;
   LoadsVoltageBalanceEventFail : ALIAS FOR DINT00_32.6;
   LoadsVoltageBalanceEventSuccess : ALIAS FOR DINT00_32.7;
   LoadsVoltageBalanceFailTimer : ALIAS FOR CLTIMER00_90;
   LoadsVoltageBalanceInProcess : ALIAS FOR DINT00_32.8;
   LoadsVoltageBalanceMsg : ALIAS FOR MESSAGE00_23;
   LoadsVoltageBalanceSuccessTimer : ALIAS FOR CLTIMER00_91;
   LoadsvoltageHILS : ALIAS FOR plc1_local_5[1];
   LoadsvoltageRaw : ALIAS FOR Local:1:I.Ch8Data;
   LoadsVoltageRebalancedEventFail : ALIAS FOR DINT00_32.9;
   LoadsVoltageRebalancedEventSuccess : ALIAS FOR DINT00_32.10;
   LoadsVoltageRebalancedFailTimer : ALIAS FOR CLTIMER00_92;
   LoadsVoltageRebalancedInProcess : ALIAS FOR DINT00_32.11;
   LoadsVoltageRebalancedMsg : ALIAS FOR MESSAGE00_24;
   LoadsVoltageRebalancedSuccessTimer : ALIAS FOR CLTIMER00_93;
   MESSAGE00_0 : MESSAGE;
        MessageParameters(ServiceCode := 16#0035, LocalElement := MESSAGE00_0_S[0], DestinationTag := MESSAGE00_0_R[0], ...)
   MESSAGE00_0_R : STRING[2] := ([0] := '                                                                                  ', [1] := '                                                              ');
   MESSAGE00_0_S : STRING[2] := ([0] := '<EVENT NAME="$$StorageManagement.SOCTooLow" DEST="Battery" SUCCESS="BatterySOCTooLo', [1] := 'wEventSuccess" FAILURE="BatterySOCTooLowEventFail"/>');
   MESSAGE00_1 : MESSAGE;
        MessageParameters(ServiceCode := 16#0035, LocalElement := MESSAGE00_1_S[0], DestinationTag := MESSAGE00_1_R[0], ...)
   MESSAGE00_10 : MESSAGE;
        MessageParameters(ServiceCode := 16#0035, LocalElement := MESSAGE00_10_S[0], DestinationTag := MESSAGE00_10_R[0], ...)
   MESSAGE00_10_R : STRING[2] := ([0] := '                                                                                  ', [1] := '                                                                      ');
   MESSAGE00_10_S : STRING[2] := ([0] := '<EVENT NAME="$$PowerManagement.PurchasePower" DEST="Load05" SUCCESS="Load05Purchase', [1] := 'PowerEventSuccess" FAILURE="Load05PurchasePowerEventFail"/>');
   MESSAGE00_11 : MESSAGE;
        MessageParameters(ServiceCode := 16#0035, LocalElement := MESSAGE00_11_S[0], DestinationTag := MESSAGE00_11_R[0], ...)
   MESSAGE00_11_R : STRING[3] := ([0] := '                                                                                  ', [1] := '                                                                                  ', [2] := '    ');
   MESSAGE00_11_S : STRING[2] := ([0] := '<EVENT NAME="$$StreetManagement.OverCurrentCondition" DEST="Comm" SUCCESS="CommOver', [1] := 'CurrentConditionEventSuccess" FAILURE="CommOverCurrentConditionEventFail"/>');
   MESSAGE00_12 : MESSAGE;
        MessageParameters(ServiceCode := 16#0035, LocalElement := MESSAGE00_12_S[0], DestinationTag := MESSAGE00_12_R[0], ...)
   MESSAGE00_12_R : STRING[2] := ([0] := '                                                                                  ', [1] := '                                                                              ');
   MESSAGE00_12_S : STRING[2] := ([0] := '<EVENT NAME="$$PowerManagement.DisconnectPower" DEST="House01" SUCCESS="House01Disc', [1] := 'onnectPowerEventSuccess" FAILURE="House01DisconnectPowerEventFail"/>');
   MESSAGE00_13 : MESSAGE;
        MessageParameters(ServiceCode := 16#0035, LocalElement := MESSAGE00_13_S[0], DestinationTag := MESSAGE00_13_R[0], ...)
   MESSAGE00_13_R : STRING[2] := ([0] := '                                                                                  ', [1] := '                                                                        ');
   MESSAGE00_13_S : STRING[2] := ([0] := '<EVENT NAME="$$PowerManagement.PurchasePower" DEST="House01" SUCCESS="House01Purcha', [1] := 'sePowerEventSuccess" FAILURE="House01PurchasePowerEventFail"/>');
   MESSAGE00_14 : MESSAGE;
        MessageParameters(ServiceCode := 16#0035, LocalElement := MESSAGE00_14_S[0], DestinationTag := MESSAGE00_14_R[0], ...)
   MESSAGE00_14_R : STRING[2] := ([0] := '                                                                                  ', [1] := '                                                                              ');
   MESSAGE00_14_S : STRING[2] := ([0] := '<EVENT NAME="$$PowerManagement.DisconnectPower" DEST="House02" SUCCESS="House02Disc', [1] := 'onnectPowerEventSuccess" FAILURE="House02DisconnectPowerEventFail"/>');
   MESSAGE00_15 : MESSAGE;
        MessageParameters(ServiceCode := 16#0035, LocalElement := MESSAGE00_15_S[0], DestinationTag := MESSAGE00_15_R[0], ...)
   MESSAGE00_15_R : STRING[2] := ([0] := '                                                                                  ', [1] := '                                                                        ');
   MESSAGE00_15_S : STRING[2] := ([0] := '<EVENT NAME="$$PowerManagement.PurchasePower" DEST="House02" SUCCESS="House02Purcha', [1] := 'sePowerEventSuccess" FAILURE="House02PurchasePowerEventFail"/>');
   MESSAGE00_16 : MESSAGE;
        MessageParameters(ServiceCode := 16#0035, LocalElement := MESSAGE00_16_S[0], DestinationTag := MESSAGE00_16_R[0], ...)
   MESSAGE00_16_R : STRING[2] := ([0] := '                                                                                  ', [1] := '                                                                              ');
   MESSAGE00_16_S : STRING[2] := ([0] := '<EVENT NAME="$$PowerManagement.DisconnectPower" DEST="House03" SUCCESS="House03Disc', [1] := 'onnectPowerEventSuccess" FAILURE="House03DisconnectPowerEventFail"/>');
   MESSAGE00_17 : MESSAGE;
        MessageParameters(ServiceCode := 16#0035, LocalElement := MESSAGE00_17_S[0], DestinationTag := MESSAGE00_17_R[0], ...)
   MESSAGE00_17_R : STRING[2] := ([0] := '                                                                                  ', [1] := '                                                                        ');
   MESSAGE00_17_S : STRING[2] := ([0] := '<EVENT NAME="$$PowerManagement.PurchasePower" DEST="House03" SUCCESS="House03Purcha', [1] := 'sePowerEventSuccess" FAILURE="House03PurchasePowerEventFail"/>');
   MESSAGE00_18 : MESSAGE;
        MessageParameters(ServiceCode := 16#0035, LocalElement := MESSAGE00_18_S[0], DestinationTag := MESSAGE00_18_R[0], ...)
   MESSAGE00_18_R : STRING[2] := ([0] := '                                                                                  ', [1] := '                                                                              ');
   MESSAGE00_18_S : STRING[2] := ([0] := '<EVENT NAME="$$PowerManagement.DisconnectPower" DEST="House04" SUCCESS="House04Disc', [1] := 'onnectPowerEventSuccess" FAILURE="House04DisconnectPowerEventFail"/>');
   MESSAGE00_19 : MESSAGE;
        MessageParameters(ServiceCode := 16#0035, LocalElement := MESSAGE00_19_S[0], DestinationTag := MESSAGE00_19_R[0], ...)
   MESSAGE00_19_R : STRING[2] := ([0] := '                                                                                  ', [1] := '                                                                        ');
   MESSAGE00_19_S : STRING[2] := ([0] := '<EVENT NAME="$$PowerManagement.PurchasePower" DEST="House04" SUCCESS="House04Purcha', [1] := 'sePowerEventSuccess" FAILURE="House04PurchasePowerEventFail"/>');
   MESSAGE00_1_R : STRING[2] := ([0] := '                                                                                  ', [1] := '                                                                            ');
   MESSAGE00_1_S : STRING[2] := ([0] := '<EVENT NAME="$$PowerManagement.DisconnectPower" DEST="Load01" SUCCESS="Load01Discon', [1] := 'nectPowerEventSuccess" FAILURE="Load01DisconnectPowerEventFail"/>');
   MESSAGE00_2 : MESSAGE;
        MessageParameters(ServiceCode := 16#0035, LocalElement := MESSAGE00_2_S[0], DestinationTag := MESSAGE00_2_R[0], ...)
   MESSAGE00_20 : MESSAGE;
        MessageParameters(ServiceCode := 16#0035, LocalElement := MESSAGE00_20_S[0], DestinationTag := MESSAGE00_20_R[0], ...)
   MESSAGE00_20_R : STRING[2] := ([0] := '                                                                                  ', [1] := '                                                                              ');
   MESSAGE00_20_S : STRING[2] := ([0] := '<EVENT NAME="$$PowerManagement.DisconnectPower" DEST="House05" SUCCESS="House05Disc', [1] := 'onnectPowerEventSuccess" FAILURE="House05DisconnectPowerEventFail"/>');
   MESSAGE00_21 : MESSAGE;
        MessageParameters(ServiceCode := 16#0035, LocalElement := MESSAGE00_21_S[0], DestinationTag := MESSAGE00_21_R[0], ...)
   MESSAGE00_21_R : STRING[2] := ([0] := '                                                                                  ', [1] := '                                                                        ');
   MESSAGE00_21_S : STRING[2] := ([0] := '<EVENT NAME="$$PowerManagement.PurchasePower" DEST="House05" SUCCESS="House05Purcha', [1] := 'sePowerEventSuccess" FAILURE="House05PurchasePowerEventFail"/>');
   MESSAGE00_22 : MESSAGE;
        MessageParameters(ServiceCode := 16#0035, LocalElement := MESSAGE00_22_S[0], DestinationTag := MESSAGE00_22_R[0], ...)
   MESSAGE00_22_R : STRING[2] := ([0] := '                                                                                  ', [1] := '                                                                                  ');
   MESSAGE00_22_S : STRING[2] := ([0] := '<EVENT NAME="$$StreetManagement.OverCurrentCondition" DEST="Res" SUCCESS="ResOverCu', [1] := 'rrentConditionEventSuccess" FAILURE="ResOverCurrentConditionEventFail"/>');
   MESSAGE00_23 : MESSAGE;
        MessageParameters(ServiceCode := 16#0035, LocalElement := MESSAGE00_23_S[0], DestinationTag := MESSAGE00_23_R[0], ...)
   MESSAGE00_23_R : STRING[2] := ([0] := '                                                                                  ', [1] := '                                                                      ');
   MESSAGE00_23_S : STRING[2] := ([0] := '<EVENT NAME="$$DistLineBalance.VoltageBalance" DEST="Loads" SUCCESS="LoadsVoltageBa', [1] := 'lanceEventSuccess" FAILURE="LoadsVoltageBalanceEventFail"/>');
   MESSAGE00_24 : MESSAGE;
        MessageParameters(ServiceCode := 16#0035, LocalElement := MESSAGE00_24_S[0], DestinationTag := MESSAGE00_24_R[0], ...)
   MESSAGE00_24_R : STRING[2] := ([0] := '                                                                                  ', [1] := '                                                                              ');
   MESSAGE00_24_S : STRING[2] := ([0] := '<EVENT NAME="$$DistLineBalance.VoltageRebalanced" DEST="Loads" SUCCESS="LoadsVoltag', [1] := 'eRebalancedEventSuccess" FAILURE="LoadsVoltageRebalancedEventFail"/>');
   MESSAGE00_25 : MESSAGE;
        MessageParameters(ServiceCode := 16#0035, LocalElement := MESSAGE00_25_S[0], DestinationTag := MESSAGE00_25_R[0], ...)
   MESSAGE00_25_R : STRING[2] := ([0] := '                                                                                  ', [1] := '                                                            ');
   MESSAGE00_25_S : STRING[2] := ([0] := '<EVENT NAME="$$GridManagement.Reset" DEST="DCMicroGrid" SUCCESS="DCMicroGridResetEv', [1] := 'entSuccess" FAILURE="DCMicroGridResetEventFail"/>');
   MESSAGE00_26 : MESSAGE;
        MessageParameters(ServiceCode := 16#0035, LocalElement := MESSAGE00_26_S[0], DestinationTag := MESSAGE00_26_R[0], ...)
   MESSAGE00_26_R : STRING[2] := ([0] := '                                                                                  ', [1] := '                                                                    ');
   MESSAGE00_26_S : STRING[2] := ([0] := '<EVENT NAME="$$GridManagement.Shutdown" DEST="DCMicroGrid" SUCCESS="DCMicroGridShut', [1] := 'downEventSuccess" FAILURE="DCMicroGridShutdownEventFail"/>');
   MESSAGE00_27 : MESSAGE;
        MessageParameters(ServiceCode := 16#0035, LocalElement := MESSAGE00_27_S[0], DestinationTag := MESSAGE00_27_R[0], ...)
   MESSAGE00_27_R : STRING[2] := ([0] := '                                                                                  ', [1] := '                                                                  ');
   MESSAGE00_27_S : STRING[2] := ([0] := '<EVENT NAME="$$GridManagement.Startup" DEST="DCMicroGrid" SUCCESS="DCMicroGridStart', [1] := 'upEventSuccess" FAILURE="DCMicroGridStartupEventFail"/>');
   MESSAGE00_28 : MESSAGE;
        MessageParameters(ServiceCode := 16#0035, LocalElement := MESSAGE00_28_S, DestinationTag := MESSAGE00_28_R, ...)
   MESSAGE00_28_R : STRING := '                                                    ';
   MESSAGE00_28_S : STRING := '<EVENT NAME="$$." DEST="" SUCCESS="" FAILURE=""/>';
   MESSAGE00_29 : MESSAGE;
        MessageParameters(ServiceCode := 16#0035, LocalElement := MESSAGE00_29_S, DestinationTag := MESSAGE00_29_R, ...)
   MESSAGE00_29_R : STRING := '                                                    ';
   MESSAGE00_29_S : STRING := '<EVENT NAME="$$." DEST="" SUCCESS="" FAILURE=""/>';
   MESSAGE00_2_R : STRING[2] := ([0] := '                                                                                  ', [1] := '                                                                      ');
   MESSAGE00_2_S : STRING[2] := ([0] := '<EVENT NAME="$$PowerManagement.PurchasePower" DEST="Load01" SUCCESS="Load01Purchase', [1] := 'PowerEventSuccess" FAILURE="Load01PurchasePowerEventFail"/>');
   MESSAGE00_3 : MESSAGE;
        MessageParameters(ServiceCode := 16#0035, LocalElement := MESSAGE00_3_S[0], DestinationTag := MESSAGE00_3_R[0], ...)
   MESSAGE00_30 : MESSAGE;
        MessageParameters(ServiceCode := 16#0035, LocalElement := MESSAGE00_30_S, DestinationTag := MESSAGE00_30_R, ...)
   MESSAGE00_30_R : STRING := '                                                    ';
   MESSAGE00_30_S : STRING := '<EVENT NAME="$$." DEST="" SUCCESS="" FAILURE=""/>';
   MESSAGE00_31 : MESSAGE;
        MessageParameters(ServiceCode := 16#0035, LocalElement := MESSAGE00_31_S, DestinationTag := MESSAGE00_31_R, ...)
   MESSAGE00_31_R : STRING := '                                                    ';
   MESSAGE00_31_S : STRING := '<EVENT NAME="$$." DEST="" SUCCESS="" FAILURE=""/>';
   MESSAGE00_32 : MESSAGE;
        MessageParameters(ServiceCode := 16#0035, LocalElement := MESSAGE00_32_S, DestinationTag := MESSAGE00_32_R, ...)
   MESSAGE00_32_R : STRING := '                                                    ';
   MESSAGE00_32_S : STRING := '<EVENT NAME="$$." DEST="" SUCCESS="" FAILURE=""/>';
   MESSAGE00_3_R : STRING[2] := ([0] := '                                                                                  ', [1] := '                                                                            ');
   MESSAGE00_3_S : STRING[2] := ([0] := '<EVENT NAME="$$PowerManagement.DisconnectPower" DEST="Load02" SUCCESS="Load02Discon', [1] := 'nectPowerEventSuccess" FAILURE="Load02DisconnectPowerEventFail"/>');
   MESSAGE00_4 : MESSAGE;
        MessageParameters(ServiceCode := 16#0035, LocalElement := MESSAGE00_4_S[0], DestinationTag := MESSAGE00_4_R[0], ...)
   MESSAGE00_4_R : STRING[2] := ([0] := '                                                                                  ', [1] := '                                                                      ');
   MESSAGE00_4_S : STRING[2] := ([0] := '<EVENT NAME="$$PowerManagement.PurchasePower" DEST="Load02" SUCCESS="Load02Purchase', [1] := 'PowerEventSuccess" FAILURE="Load02PurchasePowerEventFail"/>');
   MESSAGE00_5 : MESSAGE;
        MessageParameters(ServiceCode := 16#0035, LocalElement := MESSAGE00_5_S[0], DestinationTag := MESSAGE00_5_R[0], ...)
   MESSAGE00_5_R : STRING[2] := ([0] := '                                                                                  ', [1] := '                                                                            ');
   MESSAGE00_5_S : STRING[2] := ([0] := '<EVENT NAME="$$PowerManagement.DisconnectPower" DEST="Load03" SUCCESS="Load03Discon', [1] := 'nectPowerEventSuccess" FAILURE="Load03DisconnectPowerEventFail"/>');
   MESSAGE00_6 : MESSAGE;
        MessageParameters(ServiceCode := 16#0035, LocalElement := MESSAGE00_6_S[0], DestinationTag := MESSAGE00_6_R[0], ...)
   MESSAGE00_6_R : STRING[2] := ([0] := '                                                                                  ', [1] := '                                                                      ');
   MESSAGE00_6_S : STRING[2] := ([0] := '<EVENT NAME="$$PowerManagement.PurchasePower" DEST="Load03" SUCCESS="Load03Purchase', [1] := 'PowerEventSuccess" FAILURE="Load03PurchasePowerEventFail"/>');
   MESSAGE00_7 : MESSAGE;
        MessageParameters(ServiceCode := 16#0035, LocalElement := MESSAGE00_7_S[0], DestinationTag := MESSAGE00_7_R[0], ...)
   MESSAGE00_7_R : STRING[2] := ([0] := '                                                                                  ', [1] := '                                                                            ');
   MESSAGE00_7_S : STRING[2] := ([0] := '<EVENT NAME="$$PowerManagement.DisconnectPower" DEST="Load04" SUCCESS="Load04Discon', [1] := 'nectPowerEventSuccess" FAILURE="Load04DisconnectPowerEventFail"/>');
   MESSAGE00_8 : MESSAGE;
        MessageParameters(ServiceCode := 16#0035, LocalElement := MESSAGE00_8_S[0], DestinationTag := MESSAGE00_8_R[0], ...)
   MESSAGE00_8_R : STRING[2] := ([0] := '                                                                                  ', [1] := '                                                                      ');
   MESSAGE00_8_S : STRING[2] := ([0] := '<EVENT NAME="$$PowerManagement.PurchasePower" DEST="Load04" SUCCESS="Load04Purchase', [1] := 'PowerEventSuccess" FAILURE="Load04PurchasePowerEventFail"/>');
   MESSAGE00_9 : MESSAGE;
        MessageParameters(ServiceCode := 16#0035, LocalElement := MESSAGE00_9_S[0], DestinationTag := MESSAGE00_9_R[0], ...)
   MESSAGE00_9_R : STRING[2] := ([0] := '                                                                                  ', [1] := '                                                                            ');
   MESSAGE00_9_S : STRING[2] := ([0] := '<EVENT NAME="$$PowerManagement.DisconnectPower" DEST="Load05" SUCCESS="Load05Discon', [1] := 'nectPowerEventSuccess" FAILURE="Load05DisconnectPowerEventFail"/>');
   plc1_local_1 : REAL[10];
   plc1_local_2 : REAL[10] := ([0] := 1.1582979e-05, [1] := 1.1582978e-05, [2] := 1.1582979e-05, [3] := 1.1582978e-05, [4] := 1.1582979e-05, [5] := 1.1583727e-05, [6] := 1.1583727e-05, [7] := 1.15837265e-05, [8] := 1.15837265e-05, [9] := 1.15837265e-05);
   plc1_local_3 : REAL[10] := ([0] := 8.2350445e-05, [1] := 12.0, [2] := 0.00011963654, [3] := 12.0, [4] := 5.0513023e-05, [5] := 11.99989, [6] := 6.3704996e-05, [7] := 0.57970494, [8] := 6.3709806e-05, [9] := 0.5794644);
   plc1_local_5 : REAL[10] := ([0] := 0.0001274148, [1] := 3.7649548);
   plc1_local_6 : DINT[10];
   PricedecreaseInProcess : BOOL := 1;
   PriceDecreaseTimer : TIMER := (PRE := 5000);
   PriceIncreaseTimer : TIMER := (PRE := 5000);
   PriorityDecreaseInProcess : BOOL := 1;
   PriorityDecreaseTimer : TIMER := (PRE := 5000);
   PriorityIncreaseTimer : TIMER := (PRE := 5000);
   RB_SG1_Relay : ALIAS FOR plc1_local_6[1].2;
   RB_SG2_Relay : ALIAS FOR plc1_local_6[1].3;
   REAL00_0 : REAL := 0.25061035;
   REAL00_1 : REAL := 2.883545;
   REAL00_10 : REAL := 0.99118096;
   REAL00_100 : REAL := 1.5268278;
   REAL00_101 : REAL := 72781.62;
   REAL00_102 : REAL := 8.366149e-05;
   REAL00_103 : REAL := 0.0478611;
   REAL00_104 : REAL := 0.0046920776;
   REAL00_105 : REAL := 0.017455101;
   REAL00_106 : REAL := 0.00019674341;
   REAL00_107 : REAL := 11.0;
   REAL00_108 : REAL := 0.00027437563;
   REAL00_109 : REAL := 0.048799515;
   REAL00_11 : REAL := 0.37276268;
   REAL00_110 : REAL := 0.005;
   REAL00_111 : REAL := 1.25;
   REAL00_112 : REAL := 2.3841858e-07;
   REAL00_113 : REAL := 0.005;
   REAL00_114 : REAL := 0.048799276;
   REAL00_115 : REAL := 125.0607;
   REAL00_116 : REAL := 1.0;
   REAL00_117 : REAL := 0.016141176;
   REAL00_118 : REAL := 0.005;
   REAL00_119 : REAL := 0.001;
   REAL00_12 : REAL := 0.69118094;
   REAL00_120 : REAL := 0.0001680053;
   REAL00_121 : REAL := 125.0;
   REAL00_122 : REAL := 10.0;
   REAL00_123 : REAL := 15.0;
   REAL00_124 : REAL := 1.0;
   REAL00_125 : REAL := 10.0;
   REAL00_126 : REAL := 1.2096381;
   REAL00_127 : REAL := 103.38687;
   REAL00_128 : REAL := 1111.0885;
   REAL00_129 : REAL := 1.0;
   REAL00_13 : REAL := 7.0;
   REAL00_130 : REAL := 2.3841858e-07;
   REAL00_131 : REAL := 0.005;
   REAL00_132 : REAL := 0.001;
   REAL00_133 : REAL := 0.00011600057;
   REAL00_134 : REAL := 1111.0;
   REAL00_135 : REAL := 10.0;
   REAL00_136 : REAL := 15.0;
   REAL00_137 : REAL := 1.0;
   REAL00_138 : REAL := 10.0;
   REAL00_139 : REAL := 0.8352041;
   REAL00_14 : REAL := 0.13999999;
   REAL00_140 : REAL := 1330.3197;
   REAL00_141 : REAL := 1111.0908;
   REAL00_142 : REAL := 1.0;
   REAL00_143 : REAL := 0.016328812;
   REAL00_144 : REAL := 0.005;
   REAL00_145 : REAL := 0.001;
   REAL00_146 : REAL := 0.00015145242;
   REAL00_147 : REAL := 1111.0;
   REAL00_148 : REAL := 10.0;
   REAL00_149 : REAL := 15.0;
   REAL00_15 : REAL := 0.28479385;
   REAL00_150 : REAL := 1.0;
   REAL00_151 : REAL := 10.0;
   REAL00_152 : REAL := 1.0904574;
   REAL00_153 : REAL := 1018.92175;
   REAL00_154 : REAL := 1111111.0;
   REAL00_155 : REAL := 1.0;
   REAL00_156 : REAL := 2.3841858e-07;
   REAL00_157 : REAL := 0.005;
   REAL00_158 : REAL := 0.001;
   REAL00_159 : REAL := 0.00010831091;
   REAL00_16 : REAL := 0.0026725498;
   REAL00_160 : REAL := 1111111.0;
   REAL00_161 : REAL := 10.0;
   REAL00_162 : REAL := 15.0;
   REAL00_163 : REAL := 1.0;
   REAL00_164 : REAL := 10.0;
   REAL00_165 : REAL := 0.77983856;
   REAL00_166 : REAL := 1424796.1;
   REAL00_167 : REAL := 111111.0;
   REAL00_168 : REAL := 1.0;
   REAL00_169 : REAL := 0.016422749;
   REAL00_17 : REAL := 0.009384155;
   REAL00_170 : REAL := 0.005;
   REAL00_171 : REAL := 0.001;
   REAL00_172 : REAL := 0.000401179;
   REAL00_173 : REAL := 111111.0;
   REAL00_174 : REAL := 10.0;
   REAL00_175 : REAL := 15.0;
   REAL00_176 : REAL := 1.0;
   REAL00_177 : REAL := 10.0;
   REAL00_178 : REAL := 2.8884888;
   REAL00_179 : REAL := 38466.83;
   REAL00_18 : REAL := 0.00024414062;
   REAL00_180 : REAL := 2.237357e-10;
   REAL00_181 : REAL := 0.048799515;
   REAL00_182 : REAL := 0.0009384155;
   REAL00_183 : REAL := 8.3222076e-05;
   REAL00_184 : REAL := 0.015718937;
   REAL00_185 : REAL := 100.0;
   REAL00_186 : REAL := 10.0;
   REAL00_187 : REAL := 0.017830372;
   REAL00_188 : REAL := 0.005;
   REAL00_189 : REAL := 60.0;
   REAL00_19 : REAL := 30.0;
   REAL00_190 : REAL := 0.0005814558;
   REAL00_191 : REAL := 0.032610416;
   REAL00_192 : REAL;
   REAL00_193 : REAL := -inf;
   REAL00_194 : REAL;
   REAL00_195 : REAL;
   REAL00_196 : REAL;
   REAL00_197 : REAL;
   REAL00_198 : REAL;
   REAL00_199 : REAL;
   REAL00_2 : REAL := 11.506088;
   REAL00_20 : REAL := 1.1847997;
   REAL00_200 : REAL;
   REAL00_201 : REAL;
   REAL00_202 : REAL;
   REAL00_203 : REAL;
   REAL00_204 : REAL;
   REAL00_205 : REAL;
   REAL00_206 : REAL;
   REAL00_207 : REAL;
   REAL00_208 : REAL;
   REAL00_209 : REAL;
   REAL00_21 : REAL := 0.35;
   REAL00_210 : REAL;
   REAL00_211 : REAL;
   REAL00_212 : REAL;
   REAL00_213 : REAL;
   REAL00_214 : REAL;
   REAL00_215 : REAL;
   REAL00_216 : REAL;
   REAL00_217 : REAL;
   REAL00_218 : REAL;
   REAL00_219 : REAL;
   REAL00_22 : REAL := 11.877472;
   REAL00_220 : REAL;
   REAL00_221 : REAL;
   REAL00_222 : REAL;
   REAL00_223 : REAL;
   REAL00_224 : REAL;
   REAL00_225 : REAL;
   REAL00_226 : REAL;
   REAL00_227 : REAL;
   REAL00_228 : REAL;
   REAL00_229 : REAL;
   REAL00_23 : REAL := 0.1997;
   REAL00_230 : REAL;
   REAL00_231 : REAL;
   REAL00_24 : REAL := 12.372763;
   REAL00_25 : REAL := 99.118095;
   REAL00_26 : REAL := 69.118095;
   REAL00_27 : REAL := 0.2699999;
   REAL00_28 : REAL := 4.9911313;
   REAL00_29 : REAL := 10.0;
   REAL00_3 : REAL := 6.9382668;
   REAL00_30 : REAL := 8.3222076e-05;
   REAL00_31 : REAL := 0.0478611;
   REAL00_32 : REAL := 0.005;
   REAL00_33 : REAL := 2.5;
   REAL00_34 : REAL := 0.017830372;
   REAL00_35 : REAL := 0.005;
   REAL00_36 : REAL := 0.030124426;
   REAL00_37 : REAL := 11111.056;
   REAL00_38 : REAL := 1.0;
   REAL00_39 : REAL := 0.015859604;
   REAL00_4 : REAL;
   REAL00_40 : REAL := 0.005;
   REAL00_41 : REAL := 0.001;
   REAL00_42 : REAL := 0.00021961895;
   REAL00_43 : REAL := 11111.0;
   REAL00_44 : REAL := 10.0;
   REAL00_45 : REAL := 15.0;
   REAL00_46 : REAL := 1.0;
   REAL00_47 : REAL := 10.0;
   REAL00_48 : REAL := 1.5812564;
   REAL00_49 : REAL := 7026.726;
   REAL00_5 : REAL := 4.8382664;
   REAL00_50 : REAL := 11124.569;
   REAL00_51 : REAL := 1.0;
   REAL00_52 : REAL := 2.3841858e-07;
   REAL00_53 : REAL := 0.005;
   REAL00_54 : REAL := 0.001;
   REAL00_55 : REAL := 0.00017230643;
   REAL00_56 : REAL := 11125.0;
   REAL00_57 : REAL := 10.0;
   REAL00_58 : REAL := 15.0;
   REAL00_59 : REAL := 1.0;
   REAL00_6 : REAL := 0.00026927018;
   REAL00_60 : REAL := 10.0;
   REAL00_61 : REAL := 1.2406063;
   REAL00_62 : REAL := 8967.042;
   REAL00_63 : REAL := 1124.237;
   REAL00_64 : REAL := 1.0;
   REAL00_65 : REAL := 0.015859604;
   REAL00_66 : REAL := 0.005;
   REAL00_67 : REAL := 0.001;
   REAL00_68 : REAL := 0.00022261673;
   REAL00_69 : REAL := 1125.0;
   REAL00_7 : REAL := 0.9693727;
   REAL00_70 : REAL := 10.0;
   REAL00_71 : REAL := 15.0;
   REAL00_72 : REAL := 1.0;
   REAL00_73 : REAL := 10.0;
   REAL00_74 : REAL := 1.6028404;
   REAL00_75 : REAL := 701.403;
   REAL00_76 : REAL := 11124.747;
   REAL00_77 : REAL := 1.0;
   REAL00_78 : REAL := 2.3841858e-07;
   REAL00_79 : REAL := 0.005;
   REAL00_8 : REAL := 0.95;
   REAL00_80 : REAL := 0.001;
   REAL00_81 : REAL := 0.00016943911;
   REAL00_82 : REAL := 11125.0;
   REAL00_83 : REAL := 10.0;
   REAL00_84 : REAL := 15.0;
   REAL00_85 : REAL := 1.0;
   REAL00_86 : REAL := 10.0;
   REAL00_87 : REAL := 1.2199616;
   REAL00_88 : REAL := 9118.932;
   REAL00_89 : REAL := 111125.0;
   REAL00_9 : REAL := 2.337641;
   REAL00_90 : REAL := 1.0;
   REAL00_91 : REAL := 0.016235113;
   REAL00_92 : REAL := 0.005;
   REAL00_93 : REAL := 0.001;
   REAL00_94 : REAL := 0.00021205941;
   REAL00_95 : REAL := 111125.0;
   REAL00_96 : REAL := 10.0;
   REAL00_97 : REAL := 15.0;
   REAL00_98 : REAL := 1.0;
   REAL00_99 : REAL := 10.0;
   Resaccum : ALIAS FOR REAL00_109;
   ResBattempt : ALIAS FOR DINT00_10;
   ResBclose : ALIAS FOR Local:3:O.Data.10;
   ResBcloseHILS : ALIAS FOR plc1_local_6[0].10;
   ResBcloseProxy : ALIAS FOR DINT00_27.25;
   ResBdeadBand : ALIAS FOR REAL00_110;
   ResBfailedToOpen : ALIAS FOR DINT00_27.26;
   ResBintForceOpen : ALIAS FOR DINT00_27.27;
   ResBintReqClose : ALIAS FOR DINT00_27.28;
   ResBisClosed : ALIAS FOR DINT00_27.29;
   ResBisOpen : ALIAS FOR DINT00_27.30;
   ResBmaxAttempts : ALIAS FOR DINT00_11;
   ResBmaxLoadCurrent : ALIAS FOR REAL00_111;
   ResBopenTimer : ALIAS FOR CLTIMER00_48;
   ResBreqClose : ALIAS FOR DINT00_27.31;
   ResBreqOpen : ALIAS FOR DINT00_28.0;
   ResBreqReset : ALIAS FOR DINT00_28.1;
   ResBretriesFailed : ALIAS FOR DINT00_28.2;
   ResBtooMuchCurrent : ALIAS FOR DINT00_28.3;
   ResBunexpectedLowCurrent : ALIAS FOR DINT00_28.4;
   RescanNotifyUser : ALIAS FOR DINT00_28.5;
   RescommandChanged : ALIAS FOR DINT00_28.6;
   RescommandChangedTimer : ALIAS FOR CLTIMER00_49;
   Rescurrent : ALIAS FOR REAL00_112;
   RescurrentHILS : ALIAS FOR plc1_local_3[6];
   RescurrentRaw : ALIAS FOR Local:1:I.Ch11Data;
   Resdeadband : ALIAS FOR REAL00_113;
   Resdifference : ALIAS FOR REAL00_114;
   ResfailedToConnect : ALIAS FOR DINT00_28.7;
   ResfailedToDisconnect : ALIAS FOR DINT00_28.8;
   ResintReqConnect : ALIAS FOR DINT00_31.23;
   ResisConnected : ALIAS FOR DINT00_31.24;
   ResisDisconnected : ALIAS FOR DINT00_31.25;
   ResnotificationTimer : ALIAS FOR CLTIMER00_85;
   ResOverCurrentConditionEventFail : ALIAS FOR DINT00_31.26;
   ResOverCurrentConditionEventSuccess : ALIAS FOR DINT00_31.27;
   ResOverCurrentConditionFailTimer : ALIAS FOR CLTIMER00_86;
   ResOverCurrentConditionInProcess : ALIAS FOR DINT00_31.28;
   ResOverCurrentConditionMsg : ALIAS FOR MESSAGE00_22;
   ResOverCurrentConditionSuccessTimer : ALIAS FOR CLTIMER00_87;
   Respower : ALIAS FOR REAL00_180;
   ResreqConnect : ALIAS FOR DINT00_31.29;
   ResreqDisconnect : ALIAS FOR DINT00_31.30;
   RessampleNow : ALIAS FOR DINT00_31.31;
   RessampleTimer : ALIAS FOR CLTIMER00_88;
   Ressuperuser : ALIAS FOR STRING00_11;
   Restotal : ALIAS FOR REAL00_181;
   RestotalTooLarge : ALIAS FOR DINT00_32.0;
   RestotalTooSmall : ALIAS FOR DINT00_32.1;
   ResuserNotified : ALIAS FOR DINT00_32.2;
   Resvoltage : ALIAS FOR REAL00_182;
   ResvoltageHILS : ALIAS FOR plc1_local_3[7];
   ResvoltageRaw : ALIAS FOR Local:2:I.Ch1Data;
   RF_SG_Relay : ALIAS FOR plc1_local_6[1].4;
   RL1_SG1_Relay : ALIAS FOR plc1_local_6[1].8;
   RL1_SG2_Relay : ALIAS FOR plc1_local_6[1].9;
   RL2_SG1_Relay : ALIAS FOR plc1_local_6[1].10;
   RL2_SG2_Relay : ALIAS FOR plc1_local_6[1].11;
   RL3_SG1_Relay : ALIAS FOR plc1_local_6[1].12;
   RL3_SG2_Relay : ALIAS FOR plc1_local_6[1].13;
   RL4_SG1_Relay : ALIAS FOR plc1_local_6[1].14;
   RL4_SG2_Relay : ALIAS FOR plc1_local_6[1].15;
   RL5_SG1_Relay : ALIAS FOR plc1_local_6[1].16;
   RL5_SG2_Relay : ALIAS FOR plc1_local_6[1].17;
   Solar_Power : ALIAS FOR plc1_local_1[0];
   SolarMeasureTimer : TIMER := (PRE := 5000, ACC := 3911, EN := 1, TT := 1);
   SolarPanelBclose : ALIAS FOR Local:3:O.Data.13;
   SolarPanelBcloseHILS : ALIAS FOR plc1_local_6[0].12;
   SolarPanelBcloseProxy : ALIAS FOR DINT00_32.22;
   SolarPanelBintReqClose : ALIAS FOR DINT00_32.23;
   SolarPanelBisClosed : ALIAS FOR DINT00_32.24;
   SolarPanelBisOpen : ALIAS FOR DINT00_32.25;
   SolarPanelBreqClose : ALIAS FOR DINT00_32.26;
   SolarPanelBreqOpen : ALIAS FOR DINT00_32.27;
   SolarPanelcanSupplyPower : ALIAS FOR DINT00_32.28;
   SolarPanelcommandChanged : ALIAS FOR DINT00_32.29;
   SolarPanelcommandChangedTimer : ALIAS FOR CLTIMER00_99;
   SolarPanelcurrent : ALIAS FOR REAL00_187;
   SolarPanelcurrentHILS : ALIAS FOR plc1_local_3[0];
   SolarPanelcurrentRaw : ALIAS FOR Local:1:I.Ch2Data;
   SolarPaneldeadband : ALIAS FOR REAL00_188;
   SolarPanelfailedToConnect : ALIAS FOR DINT00_32.30;
   SolarPanelfailedToDisconnect : ALIAS FOR DINT00_32.31;
   SolarPanelintReqConnect : ALIAS FOR DINT00_33.0;
   SolarPanelisConnected : ALIAS FOR DINT00_33.1;
   SolarPanelisDisconnected : ALIAS FOR DINT00_33.2;
   SolarPanelisFunctional : ALIAS FOR DINT00_33.3;
   SolarPanelmaximumPower : ALIAS FOR REAL00_189;
   SolarPanelpower : ALIAS FOR REAL00_190;
   SolarPanelprovidingExcessPower : ALIAS FOR DINT00_33.4;
   SolarPanelreqConnect : ALIAS FOR DINT00_33.5;
   SolarPanelreqDisconnect : ALIAS FOR DINT00_33.6;
   SolarPanelvoltage : ALIAS FOR REAL00_191;
   SolarPanelvoltageHILS : ALIAS FOR plc1_local_3[1];
   SolarPanelvoltageRaw : ALIAS FOR Local:1:I.Ch1Data;
   SP_SG_Relay : ALIAS FOR plc1_local_6[1].0;
   STRING00_0 : STRING := 'DCMicroGrid';
   STRING00_1 : STRING := 'DCMicroGrid';
   STRING00_10 : STRING := 'DCMicroGrid';
   STRING00_11 : STRING := '3000#2/127.0.0.1:fpmaturana@ra.rockwell.com';
   STRING00_12 : STRING := '3000#2/10.88.58.30:rjstaron@ra.rockwell.com';
   STRING00_13 : STRING;
   STRING00_14 : STRING;
   STRING00_2 : STRING := 'DCMicroGrid';
   STRING00_3 : STRING := 'DCMicroGrid';
   STRING00_4 : STRING := 'DCMicroGrid';
   STRING00_5 : STRING := '3000#2/127.0.0.1:fpmaturana@ra.rockwell.com';
   STRING00_6 : STRING := 'DCMicroGrid';
   STRING00_7 : STRING := 'DCMicroGrid';
   STRING00_8 : STRING := 'DCMicroGrid';
   STRING00_9 : STRING := 'DCMicroGrid';
   UsingAgents : BOOL;
END_VAR
